// TIA Portal V20 program export: 7 tag tables, 10 data types, 12 data blocks, 14 code blocks (in call order from the OBs), 11 instance data blocks

VAR_GLOBAL   // PLC tag table "IO_PLC_Centralizer_PLC_Functinal_Test_1"
   In_Functional_Test_Odd AT %I100.0 : "IO_Device_Functinal_Test_Odd";
   Out_Test_Parameters_Odd AT %Q100.0 : "IO_Device_Test_Parameters_Odd";
   Voltage_Read_UInt AT %IW160 : UInt;
END_VAR

VAR_GLOBAL   // PLC tag table "IO_PLC_Centralizer_PLC_Functinal_Test_2"
   In_Functional_Test_Even AT %I300.0 : "IO_Device_Functinal_Test_Even";
   Out_Test_Parameters_Even AT %Q300.0 : "IO_Device_Test_Parameters_Even";
END_VAR

VAR_GLOBAL   // PLC tag table "IO_PLC_Centralizer_PLC_Functional_Test_Rework"
   In AT %I600.0 : "IO_Device_Functinal_Test_Rework";
   Out AT %Q600.0 : "IO_Device_Test_Parameters_Rework";
END_VAR

VAR_GLOBAL   // PLC tag table "PLC_Centralizer"
   Digital_Input_0 AT %I0.0 : Bool;
   Digital_Input_1 AT %I0.1 : Bool;
   Digital_Input_2 AT %I0.2 : Bool;
   Digital_Input_3 AT %I0.3 : Bool;
   Digital_Input_4 AT %I0.4 : Bool;
   Digital_Input_5 AT %I0.5 : Bool;
   Digital_Input_6 AT %I0.6 : Bool;
   Digital_Input_7 AT %I0.7 : Bool;
   Digital_Input_8 AT %I1.0 : Bool;
   Digital_Input_9 AT %I1.1 : Bool;
   Digital_Input_10 AT %I1.2 : Bool;
   Digital_Input_11 AT %I1.3 : Bool;
   Digital_Input_12 AT %I1.4 : Bool;
   Digital_Input_13 AT %I1.5 : Bool;
   Analogic_Input_0 AT %IW64 : Int;
   Analogic_Input_1 AT %IW66 : Int;
   Digital_Output_0 AT %Q0.0 : Bool;
   Digital_Output_1 AT %Q0.1 : Bool;
   Digital_Output_2 AT %Q0.2 : Bool;
   Digital_Output_3 AT %Q0.3 : Bool;
   Digital_Output_4 AT %Q0.4 : Bool;
   Digital_Output_5 AT %Q0.5 : Bool;
   Digital_Output_6 AT %Q0.6 : Bool;
   Digital_Output_7 AT %Q0.7 : Bool;
   Digital_Output_8 AT %Q1.0 : Bool;
   Digital_Output_9 AT %Q1.1 : Bool;
   Clock_Byte AT %MB0 : Byte;
   Clock_10Hz AT %M0.0 : Bool;
   Clock_5Hz AT %M0.1 : Bool;
   "Clock_2.5Hz" AT %M0.2 : Bool;
   Clock_2Hz AT %M0.3 : Bool;
   "Clock_1.25Hz" AT %M0.4 : Bool;
   Clock_1Hz AT %M0.5 : Bool;
   "Clock_0.625Hz" AT %M0.6 : Bool;
   "Clock_0.5Hz" AT %M0.7 : Bool;
   System_Byte AT %MB1 : Byte;
   FirstScan AT %M1.0 : Bool;
   DiagStatusUpdate AT %M1.1 : Bool;
   AlwaysTRUE AT %M1.2 : Bool;
   AlwaysFALSE AT %M1.3 : Bool;
END_VAR

VAR_GLOBAL   // PLC tag table "PLC_Centralizer_PLC_Production_And_Rework"
   In_PLC_Production_And_Rework AT %I500.0 : "IO_Device_Conveyor_Belt_Input";
   Out_PLC_Production_And_Rework AT %Q500.0 : "IO_Device_Conveyor_Belt_Ouput";
END_VAR

VAR_GLOBAL   // PLC tag table "SR-X100W_Entrace"
   Entrace_Read_Complete AT %I700.0 : Bool;
   Entrace_Read_Failure AT %I701.0 : Bool;
   Entrace_Read_Data AT %I702.0 : "SR-X100W_Read_Data";
   Entrace_Read_Request AT %Q700.0 : Bool;
   Entrace_Read_Complete_Clear AT %Q701.0 : Bool;
END_VAR

VAR_GLOBAL   // PLC tag table "SR-X100W_Exit"
   Exit_Read_Complete AT %I858.0 : Bool;
   Exit_Read_Failure AT %I859.0 : Bool;
   Exit_Read_Data AT %I860.0 : "SR-X100W_Read_Data";
   Exit_Read_Request AT %Q858.0 : Bool;
   Exit_Read_Complete_Clear AT %Q859.0 : Bool;
END_VAR

TYPE "Functional_Test"
   STRUCT
      Water_Fountain : String;
      Serial_Number : String[17];
      Panel_Number : SInt;
      Read_Electrical_Voltage : UInt;
      Read_Electrical_Current : UInt;
      Electrical_Current_Test : String[10];
      Visual_Test : String[10];
      Functional_Test : String[10];
   END_STRUCT;
END_TYPE

TYPE "IO_Device_Conveyor_Belt_Input"
   STRUCT
      Life_Trigger : Bool;
      Emergency_Stop_Release : Bool;
      Trigger_Read_Serial_Number_Entrace_Functional_Test : Bool;
      Trigger_Read_Serial_Number_Exit_Functional_Test : Bool;
      Selected_Voltage_220V : Bool;
      Selected_Voltage_127V : Bool;
      Carousel_Frequency_Inverter_Fail : Bool;
      Conveyor_Belt_Functional_Test_Inverter_Fail : Bool;
   END_STRUCT;
END_TYPE

TYPE "IO_Device_Conveyor_Belt_Ouput"
   STRUCT
      Start : Bool;
      Manual_Turn_On_Motor_Caroussel : Bool;
      Manual_Turn_On_Motor_Conveyor_Belt : Bool;
      Water_Foutain_Fail_Functional_Test : Bool;
      Select_Motor_Speed : SInt;
      Carousel_Voltage_Selection : SInt;
   END_STRUCT;
END_TYPE

TYPE "IO_Device_Functinal_Test_Even"
   STRUCT
      Life_Trigger_PLC_Functional_Test_2 : Bool;
      Star_Test_PLC_Functional_Test_2 : Bool;
      Button_PLC_Functional_Test_2 : Bool;
      Electrical_Current_Test_Approved_PLC_Functional_Test_2 : Bool;
      Visual_Test_Approved_PLC_Functional_Test_2 : Bool;
      Electrical_Current_Read_PLC_Functional_Test_2 : UInt;
      Life_Trigger_PLC_Functional_Test_4 : Bool;
      Star_Test_PLC_Functional_Test_4 : Bool;
      Button_PLC_Functional_Test_4 : Bool;
      Electrical_Current_Test_Approved_PLC_Functional_Test_4 : Bool;
      Visual_Test_Approved_PLC_Functional_Test_4 : Bool;
      Electrical_Current_Read_PLC_Functional_Test_4 : UInt;
      Life_Trigger_PLC_Functional_Test_6 : Bool;
      Star_Test_PLC_Functional_Test_6 : Bool;
      Button_PLC_Functional_Test_6 : Bool;
      Electrical_Current_Test_Approved_PLC_Functional_Test_6 : Bool;
      Visual_Test_Approved_PLC_Functional_Test_6 : Bool;
      Electrical_Current_Read_PLC_Functional_Test_6 : UInt;
      Life_Trigger_PLC_Functional_Test_8 : Bool;
      Star_Test_PLC_Functional_Test_8 : Bool;
      Button_PLC_Functional_Test_8 : Bool;
      Electrical_Current_Test_Approved_PLC_Functional_Test_8 : Bool;
      Visual_Test_Approved_PLC_Functional_Test_8 : Bool;
      Electrical_Current_Read_PLC_Functional_Test_8 : UInt;
      Life_Trigger_PLC_Functional_Test_10 : Bool;
      Star_Test_PLC_Functional_Test_10 : Bool;
      Button_PLC_Functional_Test_10 : Bool;
      Electrical_Current_Test_Approved_PLC_Functional_Test_10 : Bool;
      Visual_Test_Approved_PLC_Functional_Test_10 : Bool;
      Electrical_Current_Read_PLC_Functional_Test_10 : UInt;
      Life_Trigger_PLC_Functional_Test_12 : Bool;
      Star_Test_PLC_Functional_Test_12 : Bool;
      Button_PLC_Functional_Test_12 : Bool;
      Electrical_Current_Test_Approved_PLC_Functional_Test_12 : Bool;
      Visual_Test_Approved_PLC_Functional_Test_12 : Bool;
      Electrical_Current_Read_PLC_Functional_Test_12 : UInt;
      Life_Trigger_PLC_Functional_Test_14 : Bool;
      Star_Test_PLC_Functional_Test_14 : Bool;
      Button_PLC_Functional_Test_14 : Bool;
      Electrical_Current_Test_Approved_PLC_Functional_Test_14 : Bool;
      Visual_Test_Approved_PLC_Functional_Test_14 : Bool;
      Electrical_Current_Read_PLC_Functional_Test_14 : UInt;
      Life_Trigger_PLC_Functional_Test_16 : Bool;
      Star_Test_PLC_Functional_Test_16 : Bool;
      Button_PLC_Functional_Test_16 : Bool;
      Electrical_Current_Test_Approved_PLC_Functional_Test_16 : Bool;
      Visual_Test_Approved_PLC_Functional_Test_16 : Bool;
      Electrical_Current_Read_PLC_Functional_Test_16 : UInt;
      Life_Trigger_PLC_Functional_Test_18 : Bool;
      Star_Test_PLC_Functional_Test_18 : Bool;
      Button_PLC_Functional_Test_18 : Bool;
      Electrical_Current_Test_Approved_PLC_Functional_Test_18 : Bool;
      Visual_Test_Approved_PLC_Functional_Test_18 : Bool;
      Electrical_Current_Read_PLC_Functional_Test_18 : UInt;
      Life_Trigger_PLC_Functional_Test_20 : Bool;
      Star_Test_PLC_Functional_Test_20 : Bool;
      Button_PLC_Functional_Test_20 : Bool;
      Electrical_Current_Test_Approved_PLC_Functional_Test_20 : Bool;
      Visual_Test_Approved_PLC_Functional_Test_20 : Bool;
      Electrical_Current_Read_PLC_Functional_Test_20 : UInt;
      Life_Trigger_PLC_Functional_Test_22 : Bool;
      Star_Test_PLC_Functional_Test_22 : Bool;
      Button_PLC_Functional_Test_22 : Bool;
      Electrical_Current_Test_Approved_PLC_Functional_Test_22 : Bool;
      Visual_Test_Approved_PLC_Functional_Test_22 : Bool;
      Electrical_Current_Read_PLC_Functional_Test_22 : UInt;
      Life_Trigger_PLC_Functional_Test_24 : Bool;
      Star_Test_PLC_Functional_Test_24 : Bool;
      Button_PLC_Functional_Test_24 : Bool;
      Electrical_Current_Test_Approved_PLC_Functional_Test_24 : Bool;
      Visual_Test_Approved_PLC_Functional_Test_24 : Bool;
      Electrical_Current_Read_PLC_Functional_Test_24 : UInt;
      Life_Trigger_PLC_Functional_Test_26 : Bool;
      Star_Test_PLC_Functional_Test_26 : Bool;
      Button_PLC_Functional_Test_26 : Bool;
      Electrical_Current_Test_Approved_PLC_Functional_Test_26 : Bool;
      Visual_Test_Approved_PLC_Functional_Test_26 : Bool;
      Electrical_Current_Read_PLC_Functional_Test_26 : UInt;
      Life_Trigger_PLC_Functional_Test_28 : Bool;
      Star_Test_PLC_Functional_Test_28 : Bool;
      Button_PLC_Functional_Test_28 : Bool;
      Electrical_Current_Test_Approved_PLC_Functional_Test_28 : Bool;
      Visual_Test_Approved_PLC_Functional_Test_28 : Bool;
      Electrical_Current_Read_PLC_Functional_Test_28 : UInt;
      Life_Trigger_PLC_Functional_Test_30 : Bool;
      Star_Test_PLC_Functional_Test_30 : Bool;
      Button_PLC_Functional_Test_30 : Bool;
      Electrical_Current_Test_Approved_PLC_Functional_Test_30 : Bool;
      Visual_Test_Approved_PLC_Functional_Test_30 : Bool;
      Electrical_Current_Read_PLC_Functional_Test_30 : UInt;
   END_STRUCT;
END_TYPE

TYPE "IO_Device_Functinal_Test_Odd"
   STRUCT
      Life_Trigger_PLC_Functional_Test_1 : Bool;
      Star_Test_PLC_Functional_Test_1 : Bool;
      Button_PLC_Functional_Test_1 : Bool;
      Electrical_Current_Test_Approved_PLC_Functional_Test_1 : Bool;
      Visual_Test_Approved_PLC_Functional_Test_1 : Bool;
      Electrical_Current_Read_PLC_Functional_Test_1 : UInt;
      Life_Trigger_PLC_Functional_Test_3 : Bool;
      Star_Test_PLC_Functional_Test_3 : Bool;
      Button_PLC_Functional_Test_3 : Bool;
      Electrical_Current_Test_Approved_PLC_Functional_Test_3 : Bool;
      Visual_Test_Approved_PLC_Functional_Test_3 : Bool;
      Electrical_Current_Read_PLC_Functional_Test_3 : UInt;
      Life_Trigger_PLC_Functional_Test_5 : Bool;
      Star_Test_PLC_Functional_Test_5 : Bool;
      Button_PLC_Functional_Test_5 : Bool;
      Electrical_Current_Test_Approved_PLC_Functional_Test_5 : Bool;
      Visual_Test_Approved_PLC_Functional_Test_5 : Bool;
      Electrical_Current_Read_PLC_Functional_Test_5 : UInt;
      Life_Trigger_PLC_Functional_Test_7 : Bool;
      Star_Test_PLC_Functional_Test_7 : Bool;
      Button_PLC_Functional_Test_7 : Bool;
      Electrical_Current_Test_Approved_PLC_Functional_Test_7 : Bool;
      Visual_Test_Approved_PLC_Functional_Test_7 : Bool;
      Electrical_Current_Read_PLC_Functional_Test_7 : UInt;
      Life_Trigger_PLC_Functional_Test_9 : Bool;
      Star_Test_PLC_Functional_Test_9 : Bool;
      Button_PLC_Functional_Test_9 : Bool;
      Electrical_Current_Test_Approved_PLC_Functional_Test_9 : Bool;
      Visual_Test_Approved_PLC_Functional_Test_9 : Bool;
      Electrical_Current_Read_PLC_Functional_Test_9 : UInt;
      Life_Trigger_PLC_Functional_Test_11 : Bool;
      Star_Test_PLC_Functional_Test_11 : Bool;
      Button_PLC_Functional_Test_11 : Bool;
      Electrical_Current_Test_Approved_PLC_Functional_Test_11 : Bool;
      Visual_Test_Approved_PLC_Functional_Test_11 : Bool;
      Electrical_Current_Read_PLC_Functional_Test_11 : UInt;
      Life_Trigger_PLC_Functional_Test_13 : Bool;
      Star_Test_PLC_Functional_Test_13 : Bool;
      Button_PLC_Functional_Test_13 : Bool;
      Electrical_Current_Test_Approved_PLC_Functional_Test_13 : Bool;
      Visual_Test_Approved_PLC_Functional_Test_13 : Bool;
      Electrical_Current_Read_PLC_Functional_Test_13 : UInt;
      Life_Trigger_PLC_Functional_Test_15 : Bool;
      Star_Test_PLC_Functional_Test_15 : Bool;
      Button_PLC_Functional_Test_15 : Bool;
      Electrical_Current_Test_Approved_PLC_Functional_Test_15 : Bool;
      Visual_Test_Approved_PLC_Functional_Test_15 : Bool;
      Electrical_Current_Read_PLC_Functional_Test_15 : UInt;
      Life_Trigger_PLC_Functional_Test_17 : Bool;
      Star_Test_PLC_Functional_Test_17 : Bool;
      Button_PLC_Functional_Test_17 : Bool;
      Electrical_Current_Test_Approved_PLC_Functional_Test_17 : Bool;
      Visual_Test_Approved_PLC_Functional_Test_17 : Bool;
      Electrical_Current_Read_PLC_Functional_Test_17 : UInt;
      Life_Trigger_PLC_Functional_Test_19 : Bool;
      Star_Test_PLC_Functional_Test_19 : Bool;
      Button_PLC_Functional_Test_19 : Bool;
      Electrical_Current_Test_Approved_PLC_Functional_Test_19 : Bool;
      Visual_Test_Approved_PLC_Functional_Test_19 : Bool;
      Electrical_Current_Read_PLC_Functional_Test_19 : UInt;
      Life_Trigger_PLC_Functional_Test_21 : Bool;
      Star_Test_PLC_Functional_Test_21 : Bool;
      Button_PLC_Functional_Test_21 : Bool;
      Electrical_Current_Test_Approved_PLC_Functional_Test_21 : Bool;
      Visual_Test_Approved_PLC_Functional_Test_21 : Bool;
      Electrical_Current_Read_PLC_Functional_Test_21 : UInt;
      Life_Trigger_PLC_Functional_Test_23 : Bool;
      Star_Test_PLC_Functional_Test_23 : Bool;
      Button_PLC_Functional_Test_23 : Bool;
      Electrical_Current_Test_Approved_PLC_Functional_Test_23 : Bool;
      Visual_Test_Approved_PLC_Functional_Test_23 : Bool;
      Electrical_Current_Read_PLC_Functional_Test_23 : UInt;
      Life_Trigger_PLC_Functional_Test_25 : Bool;
      Star_Test_PLC_Functional_Test_25 : Bool;
      Button_PLC_Functional_Test_25 : Bool;
      Electrical_Current_Test_Approved_PLC_Functional_Test_25 : Bool;
      Visual_Test_Approved_PLC_Functional_Test_25 : Bool;
      Electrical_Current_Read_PLC_Functional_Test_25 : UInt;
      Life_Trigger_PLC_Functional_Test_27 : Bool;
      Star_Test_PLC_Functional_Test_27 : Bool;
      Button_PLC_Functional_Test_27 : Bool;
      Electrical_Current_Test_Approved_PLC_Functional_Test_27 : Bool;
      Visual_Test_Approved_PLC_Functional_Test_27 : Bool;
      Electrical_Current_Read_PLC_Functional_Test_27 : UInt;
      Life_Trigger_PLC_Functional_Test_29 : Bool;
      Star_Test_PLC_Functional_Test_29 : Bool;
      Button_PLC_Functional_Test_29 : Bool;
      Electrical_Current_Test_Approved_PLC_Functional_Test_29 : Bool;
      Visual_Test_Approved_PLC_Functional_Test_29 : Bool;
      Electrical_Current_Read_PLC_Functional_Test_29 : UInt;
   END_STRUCT;
END_TYPE

TYPE "IO_Device_Functinal_Test_Rework"
   STRUCT
      Life_Trigger_PLC_Functional_Test_Rework : Bool;
      Star_Test_PLC_Functional_Test_Rework : Bool;
      Button_PLC_Functional_Test_Rework : Bool;
      Electrical_Current_Test_Approved_PLC_Functional_Test_Rework : Bool;
      Visual_Test_Approved_PLC_Functional_Test_Rework : Bool;
      Electrical_Current_Read_PLC_Functional_Test_Rework : UInt;
   END_STRUCT;
END_TYPE

TYPE "IO_Device_Test_Parameters_Even"
   STRUCT
      Reset_PLC_Functional_Test_2 : Bool;
      Reset_PLC_Functional_Test_4 : Bool;
      Reset_PLC_Functional_Test_6 : Bool;
      Reset_PLC_Functional_Test_8 : Bool;
      Reset_PLC_Functional_Test_10 : Bool;
      Reset_PLC_Functional_Test_12 : Bool;
      Reset_PLC_Functional_Test_14 : Bool;
      Reset_PLC_Functional_Test_16 : Bool;
      Reset_PLC_Functional_Test_18 : Bool;
      Reset_PLC_Functional_Test_20 : Bool;
      Reset_PLC_Functional_Test_22 : Bool;
      Reset_PLC_Functional_Test_24 : Bool;
      Reset_PLC_Functional_Test_26 : Bool;
      Reset_PLC_Functional_Test_28 : Bool;
      Reset_PLC_Functional_Test_30 : Bool;
      Status : Bool;
      Voltage_Read : UInt;
      Min_Electrical_Current : UInt;
      Max_Electrical_Current : UInt;
      Time_End_Electrical_Current_Test : Time;
      Time_Start_Visual_Test : Time;
   END_STRUCT;
END_TYPE

TYPE "IO_Device_Test_Parameters_Odd"
   STRUCT
      Reset_PLC_Functional_Test_1 : Bool;
      Reset_PLC_Functional_Test_3 : Bool;
      Reset_PLC_Functional_Test_5 : Bool;
      Reset_PLC_Functional_Test_7 : Bool;
      Reset_PLC_Functional_Test_9 : Bool;
      Reset_PLC_Functional_Test_11 : Bool;
      Reset_PLC_Functional_Test_13 : Bool;
      Reset_PLC_Functional_Test_15 : Bool;
      Reset_PLC_Functional_Test_17 : Bool;
      Reset_PLC_Functional_Test_19 : Bool;
      Reset_PLC_Functional_Test_21 : Bool;
      Reset_PLC_Functional_Test_23 : Bool;
      Reset_PLC_Functional_Test_25 : Bool;
      Reset_PLC_Functional_Test_27 : Bool;
      Reset_PLC_Functional_Test_29 : Bool;
      Status : Bool;
      Voltage_Read : UInt;
      Min_Electrical_Current : UInt;
      Max_Electrical_Current : UInt;
      Time_End_Electrical_Current_Test : Time;
      Time_Start_Visual_Test : Time;
   END_STRUCT;
END_TYPE

TYPE "IO_Device_Test_Parameters_Rework"
   STRUCT
      Reset_PLC_Functional_Test_Rework : Bool;
      Status : Bool;
      Voltage_Read : UInt;
      Min_Electrical_Current : UInt;
      Max_Electrical_Current : UInt;
      Time_End_Electrical_Current_Test : Time;
      Time_Start_Visual_Test : Time;
   END_STRUCT;
END_TYPE

TYPE "SR-X100W_Read_Data"
   STRUCT
      "sr-x_100_Read_Data_1" : Char;
      "sr-x_100_Read_Data_2" : Char;
      "sr-x_100_Read_Data_3" : Char;
      "sr-x_100_Read_Data_4" : Char;
      "sr-x_100_Read_Data_5" : Char;
      "sr-x_100_Read_Data_6" : Char;
      "sr-x_100_Read_Data_7" : Char;
      "sr-x_100_Read_Data_8" : Char;
      "sr-x_100_Read_Data_9" : Char;
      "sr-x_100_Read_Data_10" : Char;
      "sr-x_100_Read_Data_11" : Char;
      "sr-x_100_Read_Data_12" : Char;
      "sr-x_100_Read_Data_13" : Char;
      "sr-x_100_Read_Data_14" : Char;
      "sr-x_100_Read_Data_15" : Char;
      "sr-x_100_Read_Data_16" : Char;
      "sr-x_100_Read_Data_17" : Char;
      "sr-x_100_Read_Data_18" : Char;
      "sr-x_100_Read_Data_19" : Char;
      "sr-x_100_Read_Data_20" : Char;
      "sr-x_100_Read_Data_21" : Char;
      "sr-x_100_Read_Data_22" : Char;
      "sr-x_100_Read_Data_23" : Char;
      "sr-x_100_Read_Data_24" : Char;
      "sr-x_100_Read_Data_25" : Char;
      "sr-x_100_Read_Data_26" : Char;
      "sr-x_100_Read_Data_27" : Char;
      "sr-x_100_Read_Data_28" : Char;
      "sr-x_100_Read_Data_29" : Char;
      "sr-x_100_Read_Data_30" : Char;
      "sr-x_100_Read_Data_31" : Char;
      "sr-x_100_Read_Data_32" : Char;
      "sr-x_100_Read_Data_33" : Char;
      "sr-x_100_Read_Data_34" : Char;
      "sr-x_100_Read_Data_35" : Char;
      "sr-x_100_Read_Data_36" : Char;
      "sr-x_100_Read_Data_37" : Char;
      "sr-x_100_Read_Data_38" : Char;
      "sr-x_100_Read_Data_39" : Char;
      "sr-x_100_Read_Data_40" : Char;
      "sr-x_100_Read_Data_41" : Char;
      "sr-x_100_Read_Data_42" : Char;
      "sr-x_100_Read_Data_43" : Char;
      "sr-x_100_Read_Data_44" : Char;
      "sr-x_100_Read_Data_45" : Char;
      "sr-x_100_Read_Data_46" : Char;
      "sr-x_100_Read_Data_47" : Char;
      "sr-x_100_Read_Data_48" : Char;
      "sr-x_100_Read_Data_49" : Char;
      "sr-x_100_Read_Data_50" : Char;
      "sr-x_100_Read_Data_51" : Char;
      "sr-x_100_Read_Data_52" : Char;
      "sr-x_100_Read_Data_53" : Char;
      "sr-x_100_Read_Data_54" : Char;
      "sr-x_100_Read_Data_55" : Char;
      "sr-x_100_Read_Data_56" : Char;
      "sr-x_100_Read_Data_57" : Char;
      "sr-x_100_Read_Data_58" : Char;
      "sr-x_100_Read_Data_59" : Char;
      "sr-x_100_Read_Data_60" : Char;
      "sr-x_100_Read_Data_61" : Char;
      "sr-x_100_Read_Data_62" : Char;
      "sr-x_100_Read_Data_63" : Char;
      "sr-x_100_Read_Data_64" : Char;
      "sr-x_100_Read_Data_65" : Char;
      "sr-x_100_Read_Data_66" : Char;
      "sr-x_100_Read_Data_67" : Char;
      "sr-x_100_Read_Data_68" : Char;
      "sr-x_100_Read_Data_69" : Char;
      "sr-x_100_Read_Data_70" : Char;
      "sr-x_100_Read_Data_71" : Char;
      "sr-x_100_Read_Data_72" : Char;
      "sr-x_100_Read_Data_73" : Char;
      "sr-x_100_Read_Data_74" : Char;
      "sr-x_100_Read_Data_75" : Char;
      "sr-x_100_Read_Data_76" : Char;
      "sr-x_100_Read_Data_77" : Char;
      "sr-x_100_Read_Data_78" : Char;
      "sr-x_100_Read_Data_79" : Char;
      "sr-x_100_Read_Data_80" : Char;
      "sr-x_100_Read_Data_81" : Char;
      "sr-x_100_Read_Data_82" : Char;
      "sr-x_100_Read_Data_83" : Char;
      "sr-x_100_Read_Data_84" : Char;
      "sr-x_100_Read_Data_85" : Char;
      "sr-x_100_Read_Data_86" : Char;
      "sr-x_100_Read_Data_87" : Char;
      "sr-x_100_Read_Data_88" : Char;
      "sr-x_100_Read_Data_89" : Char;
      "sr-x_100_Read_Data_90" : Char;
      "sr-x_100_Read_Data_91" : Char;
      "sr-x_100_Read_Data_92" : Char;
      "sr-x_100_Read_Data_93" : Char;
      "sr-x_100_Read_Data_94" : Char;
      "sr-x_100_Read_Data_95" : Char;
      "sr-x_100_Read_Data_96" : Char;
      "sr-x_100_Read_Data_97" : Char;
      "sr-x_100_Read_Data_98" : Char;
      "sr-x_100_Read_Data_99" : Char;
      "sr-x_100_Read_Data_100" : Char;
      "sr-x_100_Read_Data_101" : Char;
      "sr-x_100_Read_Data_102" : Char;
      "sr-x_100_Read_Data_103" : Char;
      "sr-x_100_Read_Data_104" : Char;
      "sr-x_100_Read_Data_105" : Char;
      "sr-x_100_Read_Data_106" : Char;
      "sr-x_100_Read_Data_107" : Char;
      "sr-x_100_Read_Data_108" : Char;
      "sr-x_100_Read_Data_109" : Char;
      "sr-x_100_Read_Data_110" : Char;
      "sr-x_100_Read_Data_111" : Char;
      "sr-x_100_Read_Data_112" : Char;
      "sr-x_100_Read_Data_113" : Char;
      "sr-x_100_Read_Data_114" : Char;
      "sr-x_100_Read_Data_115" : Char;
      "sr-x_100_Read_Data_116" : Char;
      "sr-x_100_Read_Data_117" : Char;
      "sr-x_100_Read_Data_118" : Char;
      "sr-x_100_Read_Data_119" : Char;
      "sr-x_100_Read_Data_120" : Char;
      "sr-x_100_Read_Data_121" : Char;
      "sr-x_100_Read_Data_122" : Char;
      "sr-x_100_Read_Data_123" : Char;
      "sr-x_100_Read_Data_124" : Char;
      "sr-x_100_Read_Data_125" : Char;
      "sr-x_100_Read_Data_126" : Char;
      "sr-x_100_Read_Data_127" : Char;
      "sr-x_100_Read_Data_128" : Char;
      "sr-x_100_Read_Data_129" : Char;
      "sr-x_100_Read_Data_130" : Char;
      "sr-x_100_Read_Data_131" : Char;
      "sr-x_100_Read_Data_132" : Char;
      "sr-x_100_Read_Data_133" : Char;
      "sr-x_100_Read_Data_134" : Char;
      "sr-x_100_Read_Data_135" : Char;
      "sr-x_100_Read_Data_136" : Char;
   END_STRUCT;
END_TYPE

DATA_BLOCK "DB_Analogic_Inputs"   // DB2
{ S7_Optimized_Access := 'TRUE' }
// stored: MemoryReserve 100
   VAR
      Real_Analogic_Input_0 : Real;
      Real_Analogic_Input_1 : Real;
      Uint_Analogic_Input_0 : UInt;
      Uint_Analogic_Input_1 : UInt;
   END_VAR
BEGIN
END_DATA_BLOCK

DATA_BLOCK "DB_DataLog"   // DB12
{ S7_Optimized_Access := 'TRUE' }
// stored: MemoryReserve 100
   VAR
      Create_DataLog : Bool;
      Open_DataLog : Bool;
      Write_DataLog : Bool;
      Close_DataLog : Bool;
      Clean_DataLog : Bool;
      Delete_DataLog : Bool;
      ID_DataLog : DWord;
      Name_DataLog : String := 'Teste Funcional';
      Header_DataLog : String := 'Bebedoro,Numero de Serie,Painel,Tensao Eletrica [V],Corrente Eletrica [mA],Resultado Teste Corrente,Resultado Teste Visual,Resultado Teste Funcional';
   END_VAR
BEGIN
END_DATA_BLOCK

DATA_BLOCK "DB_Digital_Inputs"   // DB1
{ S7_Optimized_Access := 'TRUE' }
// stored: MemoryReserve 100
   VAR
      Digital_Input_0 : Bool;
      Digital_Input_1 : Bool;
      Digital_Input_2 : Bool;
      Digital_Input_3 : Bool;
      Digital_Input_4 : Bool;
      Digital_Input_5 : Bool;
      Digital_Input_6 : Bool;
      Digital_Input_7 : Bool;
      Digital_Input_8 : Bool;
      Digital_Input_9 : Bool;
      Digital_Input_10 : Bool;
      Digital_Input_11 : Bool;
      Digital_Input_12 : Bool;
      Digital_Input_13 : Bool;
   END_VAR
BEGIN
END_DATA_BLOCK

DATA_BLOCK "DB_Digital_Outputs"   // DB3
{ S7_Optimized_Access := 'TRUE' }
// stored: MemoryReserve 100
   VAR
      Digital_Output_0 : Bool;
      Digital_Output_1 : Bool;
      Digital_Output_2 : Bool;
      Digital_Output_3 : Bool;
      Digital_Output_4 : Bool;
      Digital_Output_5 : Bool;
      Digital_Output_6 : Bool;
      Digital_Output_7 : Bool;
      Digital_Output_8 : Bool;
      Digital_Output_9 : Bool;
   END_VAR
BEGIN
END_DATA_BLOCK

DATA_BLOCK "DB_Found_Water_Fountain_Functional_Test"   // DB11
{ S7_Optimized_Access := 'TRUE' }
// stored: MemoryReserve 100
   VAR
      Found_Functional_Test : Bool;
      Water_Foutain_Fail_Functional_Test : Bool;
      i : SInt;
      Water_Foutain_Functional_Test : "Functional_Test";
   END_VAR
BEGIN
END_DATA_BLOCK

DATA_BLOCK "DB_HMI"   // DB4
{ S7_Optimized_Access := 'TRUE' }
// stored: MemoryReserve 100
   VAR
      Job_Mailbox : Array[0..3] of Word;
      Control_Screen : Word := 1;
      Alarm : Bool;
      Start : Bool;
      Change_Employee : Bool;
      Send_Recipe : Bool;
      Manual_Turn_On_Motor_Caroussel : Bool;
      Manual_Turn_On_Motor_Conveyor_Belt : Bool;
      Select_Test_Panel : SInt;
      Select_Motor_Speed : SInt := 1;
      Employee_Rework : String[6];
      Employee_Station_1 : String[6];
      Employee_Station_2 : String[6];
   END_VAR
   VAR RETAIN
      Admin_1 : String[6];
      Admin_2 : String[6];
      Admin_3 : String[6];
      Admin_4 : String[6];
      Admin_5 : String[6];
   END_VAR
   VAR
      Serial_Number : String[17];
      Electrical_Current : UInt;
      Electrical_Voltage : UInt;
      Electrical_Current_Result : String[10];
      Visual_Test_Result : String[10];
      Functional_Test_Result : String[10];
      Rework_Serial_Number : String[17];
      Rework_Electrical_Current : UInt;
      Rework_Electrical_Voltage : UInt;
      Rework_Electrical_Current_Result : String[10];
      Rework_Visual_Test_Result : String[10];
      Rework_Functional_Test_Result : String[10];
      Alarm_0 : Word;
      Alarm_1 : Word;
      Alarm_2 : Word;
   END_VAR
BEGIN
END_DATA_BLOCK

DATA_BLOCK "DB_IO_Device_In_Functional_Test"   // DB6
{ S7_Optimized_Access := 'TRUE' }
// stored: MemoryReserve 100
   VAR
      Reset_PLC_Functional_Test : Array[0..31] of Bool;
      Status : Bool;
      Voltage_Read : UInt;
   END_VAR
BEGIN
END_DATA_BLOCK

DATA_BLOCK "DB_IO_Device_In_Production and Rework"   // DB7
{ S7_Optimized_Access := 'TRUE' }
// stored: AutoNumber false, MemoryReserve 100
   VAR
      Emergency_Stop_Release : Bool;
      Trigger_Read_Serial_Number_Entrace_Functional_Test : Bool;
      Trigger_Read_Serial_Number_Exit_Functional_Test : Bool;
      Selected_Voltage_220V : Bool;
      Selected_Voltage_127V : Bool;
      Carousel_Frequency_Inverter_Fail : Bool;
      Conveyor_Belt_Functional_Test_Inverter_Fail : Bool;
   END_VAR
BEGIN
END_DATA_BLOCK

DATA_BLOCK "DB_Marrige"   // DB10
{ S7_Optimized_Access := 'TRUE' }
// stored: AutoNumber false, MemoryReserve 100
   VAR
      Functional_Tests_Panels : Array[0..31] of "Functional_Test";
      Got_Married { S7_SetPoint := 'True'} : Bool;
      Serial_Number : String[17];
   END_VAR
BEGIN
   Functional_Tests_Panels[0].Panel_Number := 0;
   Functional_Tests_Panels[1].Panel_Number := 1;
   Functional_Tests_Panels[2].Panel_Number := 2;
   Functional_Tests_Panels[3].Panel_Number := 3;
   Functional_Tests_Panels[4].Panel_Number := 4;
   Functional_Tests_Panels[5].Panel_Number := 5;
   Functional_Tests_Panels[6].Panel_Number := 6;
   Functional_Tests_Panels[7].Panel_Number := 7;
   Functional_Tests_Panels[8].Panel_Number := 8;
   Functional_Tests_Panels[9].Panel_Number := 9;
   Functional_Tests_Panels[10].Panel_Number := 10;
   Functional_Tests_Panels[11].Panel_Number := 11;
   Functional_Tests_Panels[12].Panel_Number := 12;
   Functional_Tests_Panels[13].Panel_Number := 13;
   Functional_Tests_Panels[14].Panel_Number := 14;
   Functional_Tests_Panels[15].Panel_Number := 15;
   Functional_Tests_Panels[16].Panel_Number := 16;
   Functional_Tests_Panels[17].Panel_Number := 17;
   Functional_Tests_Panels[18].Panel_Number := 18;
   Functional_Tests_Panels[19].Panel_Number := 19;
   Functional_Tests_Panels[20].Panel_Number := 20;
   Functional_Tests_Panels[21].Panel_Number := 21;
   Functional_Tests_Panels[22].Panel_Number := 22;
   Functional_Tests_Panels[23].Panel_Number := 23;
   Functional_Tests_Panels[24].Panel_Number := 24;
   Functional_Tests_Panels[25].Panel_Number := 25;
   Functional_Tests_Panels[26].Panel_Number := 26;
   Functional_Tests_Panels[27].Panel_Number := 27;
   Functional_Tests_Panels[28].Panel_Number := 28;
   Functional_Tests_Panels[29].Panel_Number := 29;
   Functional_Tests_Panels[30].Panel_Number := 30;
   Functional_Tests_Panels[31].Panel_Number := 31;
END_DATA_BLOCK

DATA_BLOCK "DB_Recipe"   // DB5
{ S7_Optimized_Access := 'TRUE' }
// stored: MemoryReserve 100
   VAR
      Water_Fountain : String;
      Voltage : SInt;
      Min_Electrical_Current : UInt;
      Max_Electrical_Current : UInt;
      Time_End_Electrical_Current_Test : Time;
      Time_Start_Visual_Test : Time;
   END_VAR
BEGIN
END_DATA_BLOCK

DATA_BLOCK "DB_SR-X100W_Entrace"   // DB8
{ S7_Optimized_Access := 'TRUE' }
// stored: MemoryReserve 100
   VAR
      Read_Complete_OUT : Bool;
      Read_Failure_OUT : Bool;
      Read_Data_Out : String[136];
      Serial_Number : String[17];
   END_VAR
BEGIN
END_DATA_BLOCK

DATA_BLOCK "DB_SR-X100W_Exit"   // DB9
{ S7_Optimized_Access := 'TRUE' }
// stored: AutoNumber false, MemoryReserve 100
   VAR
      Read_Complete_OUT : Bool;
      Read_Failure_OUT : Bool;
      Read_Data_Out : String[136];
      Serial_Number : String[17];
   END_VAR
BEGIN
END_DATA_BLOCK

ORGANIZATION_BLOCK "Main"   // OB1, LAD, ProgramCycle
TITLE = "Main Program Sweep (Cycle)"
{ S7_Optimized_Access := 'TRUE' }
// stored: SetENOAutomatically false
   VAR_INPUT
      Initial_Call : Bool;   // Initial call of this OB
      Remanence : Bool;   // =True, if remanent data are available
   END_VAR
BEGIN

REGION Network 1
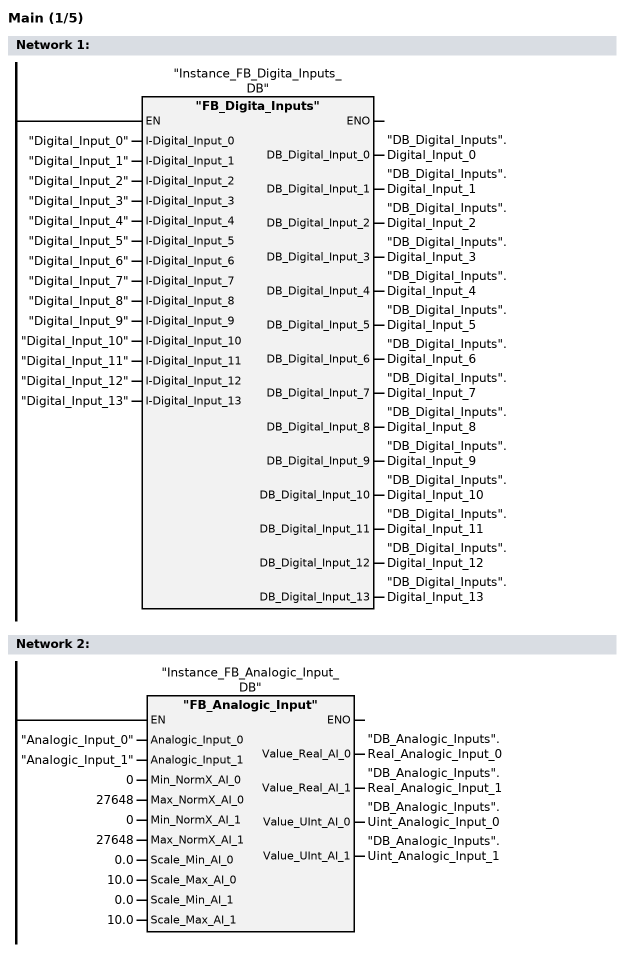
   RUNG wire#powerrail
      "Instance_FB_Digita_Inputs_DB"("I-Digital_Input_0" := "Digital_Input_0", "I-Digital_Input_1" := "Digital_Input_1", "I-Digital_Input_2" := "Digital_Input_2", "I-Digital_Input_3" := "Digital_Input_3", "I-Digital_Input_4" := "Digital_Input_4", "I-Digital_Input_5" := "Digital_Input_5", "I-Digital_Input_6" := "Digital_Input_6", "I-Digital_Input_7" := "Digital_Input_7", "I-Digital_Input_8" := "Digital_Input_8", "I-Digital_Input_9" := "Digital_Input_9", "I-Digital_Input_10" := "Digital_Input_10", "I-Digital_Input_11" := "Digital_Input_11", "I-Digital_Input_12" := "Digital_Input_12", "I-Digital_Input_13" := "Digital_Input_13", DB_Digital_Input_0 => "DB_Digital_Inputs".Digital_Input_0, DB_Digital_Input_1 => "DB_Digital_Inputs".Digital_Input_1, DB_Digital_Input_2 => "DB_Digital_Inputs".Digital_Input_2, DB_Digital_Input_3 => "DB_Digital_Inputs".Digital_Input_3, DB_Digital_Input_4 => "DB_Digital_Inputs".Digital_Input_4, DB_Digital_Input_5 => "DB_Digital_Inputs".Digital_Input_5, DB_Digital_Input_6 => "DB_Digital_Inputs".Digital_Input_6, DB_Digital_Input_7 => "DB_Digital_Inputs".Digital_Input_7, DB_Digital_Input_8 => "DB_Digital_Inputs".Digital_Input_8, DB_Digital_Input_9 => "DB_Digital_Inputs".Digital_Input_9, DB_Digital_Input_10 => "DB_Digital_Inputs".Digital_Input_10, DB_Digital_Input_11 => "DB_Digital_Inputs".Digital_Input_11, DB_Digital_Input_12 => "DB_Digital_Inputs".Digital_Input_12, DB_Digital_Input_13 => "DB_Digital_Inputs".Digital_Input_13)
   END_RUNG
   // the same network as SCL:
   "Instance_FB_Digita_Inputs_DB"("I-Digital_Input_0" := "Digital_Input_0",   // "FB_Digita_Inputs"
                           "I-Digital_Input_1" := "Digital_Input_1",
                           "I-Digital_Input_2" := "Digital_Input_2",
                           "I-Digital_Input_3" := "Digital_Input_3",
                           "I-Digital_Input_4" := "Digital_Input_4",
                           "I-Digital_Input_5" := "Digital_Input_5",
                           "I-Digital_Input_6" := "Digital_Input_6",
                           "I-Digital_Input_7" := "Digital_Input_7",
                           "I-Digital_Input_8" := "Digital_Input_8",
                           "I-Digital_Input_9" := "Digital_Input_9",
                           "I-Digital_Input_10" := "Digital_Input_10",
                           "I-Digital_Input_11" := "Digital_Input_11",
                           "I-Digital_Input_12" := "Digital_Input_12",
                           "I-Digital_Input_13" := "Digital_Input_13",
                           DB_Digital_Input_0 => "DB_Digital_Inputs".Digital_Input_0,
                           DB_Digital_Input_1 => "DB_Digital_Inputs".Digital_Input_1,
                           DB_Digital_Input_2 => "DB_Digital_Inputs".Digital_Input_2,
                           DB_Digital_Input_3 => "DB_Digital_Inputs".Digital_Input_3,
                           DB_Digital_Input_4 => "DB_Digital_Inputs".Digital_Input_4,
                           DB_Digital_Input_5 => "DB_Digital_Inputs".Digital_Input_5,
                           DB_Digital_Input_6 => "DB_Digital_Inputs".Digital_Input_6,
                           DB_Digital_Input_7 => "DB_Digital_Inputs".Digital_Input_7,
                           DB_Digital_Input_8 => "DB_Digital_Inputs".Digital_Input_8,
                           DB_Digital_Input_9 => "DB_Digital_Inputs".Digital_Input_9,
                           DB_Digital_Input_10 => "DB_Digital_Inputs".Digital_Input_10,
                           DB_Digital_Input_11 => "DB_Digital_Inputs".Digital_Input_11,
                           DB_Digital_Input_12 => "DB_Digital_Inputs".Digital_Input_12,
                           DB_Digital_Input_13 => "DB_Digital_Inputs".Digital_Input_13);
END_REGION

REGION Network 2
   RUNG wire#powerrail
      "Instance_FB_Analogic_Input_DB"(Analogic_Input_0 := "Analogic_Input_0", Analogic_Input_1 := "Analogic_Input_1", Min_NormX_AI_0 := 0, Max_NormX_AI_0 := 27648, Min_NormX_AI_1 := 0, Max_NormX_AI_1 := 27648, Scale_Min_AI_0 := 0.0, Scale_Max_AI_0 := 10.0, Scale_Min_AI_1 := 0.0, Scale_Max_AI_1 := 10.0, Value_Real_AI_0 => "DB_Analogic_Inputs".Real_Analogic_Input_0, Value_Real_AI_1 => "DB_Analogic_Inputs".Real_Analogic_Input_1, Value_UInt_AI_0 => "DB_Analogic_Inputs".Uint_Analogic_Input_0, Value_UInt_AI_1 => "DB_Analogic_Inputs".Uint_Analogic_Input_1)
   END_RUNG
   // the same network as SCL:
   "Instance_FB_Analogic_Input_DB"(Analogic_Input_0 := "Analogic_Input_0",   // "FB_Analogic_Input"
                           Analogic_Input_1 := "Analogic_Input_1",
                           Min_NormX_AI_0 := 0,
                           Max_NormX_AI_0 := 27648,
                           Min_NormX_AI_1 := 0,
                           Max_NormX_AI_1 := 27648,
                           Scale_Min_AI_0 := 0.0,
                           Scale_Max_AI_0 := 10.0,
                           Scale_Min_AI_1 := 0.0,
                           Scale_Max_AI_1 := 10.0,
                           Value_Real_AI_0 => "DB_Analogic_Inputs".Real_Analogic_Input_0,
                           Value_Real_AI_1 => "DB_Analogic_Inputs".Real_Analogic_Input_1,
                           Value_UInt_AI_0 => "DB_Analogic_Inputs".Uint_Analogic_Input_0,
                           Value_UInt_AI_1 => "DB_Analogic_Inputs".Uint_Analogic_Input_1);
END_REGION

REGION Network 3
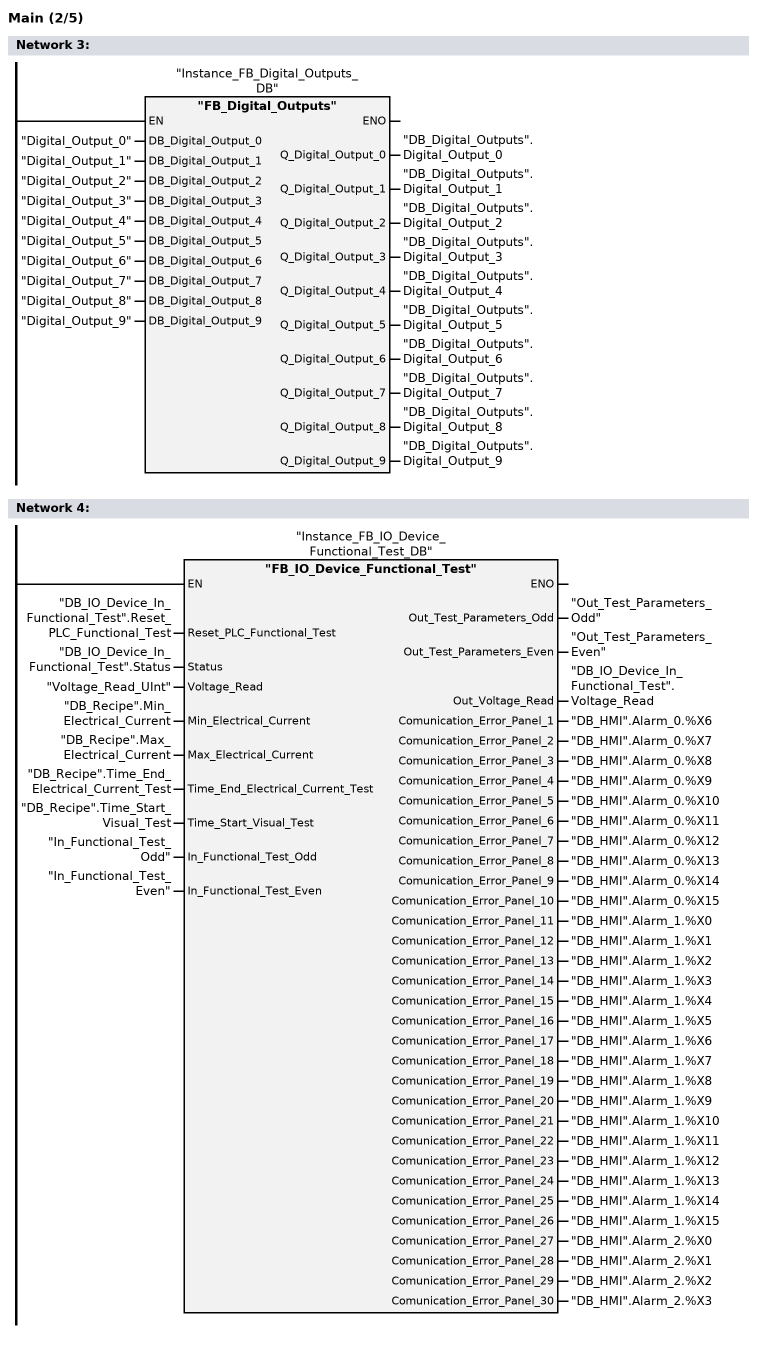
   RUNG wire#powerrail
      "Instance_FB_Digital_Outputs_DB"(DB_Digital_Output_0 := "Digital_Output_0", DB_Digital_Output_1 := "Digital_Output_1", DB_Digital_Output_2 := "Digital_Output_2", DB_Digital_Output_3 := "Digital_Output_3", DB_Digital_Output_4 := "Digital_Output_4", DB_Digital_Output_5 := "Digital_Output_5", DB_Digital_Output_6 := "Digital_Output_6", DB_Digital_Output_7 := "Digital_Output_7", DB_Digital_Output_8 := "Digital_Output_8", DB_Digital_Output_9 := "Digital_Output_9", Q_Digital_Output_0 => "DB_Digital_Outputs".Digital_Output_0, Q_Digital_Output_1 => "DB_Digital_Outputs".Digital_Output_1, Q_Digital_Output_2 => "DB_Digital_Outputs".Digital_Output_2, Q_Digital_Output_3 => "DB_Digital_Outputs".Digital_Output_3, Q_Digital_Output_4 => "DB_Digital_Outputs".Digital_Output_4, Q_Digital_Output_5 => "DB_Digital_Outputs".Digital_Output_5, Q_Digital_Output_6 => "DB_Digital_Outputs".Digital_Output_6, Q_Digital_Output_7 => "DB_Digital_Outputs".Digital_Output_7, Q_Digital_Output_8 => "DB_Digital_Outputs".Digital_Output_8, Q_Digital_Output_9 => "DB_Digital_Outputs".Digital_Output_9)
   END_RUNG
   // the same network as SCL:
   "Instance_FB_Digital_Outputs_DB"(DB_Digital_Output_0 := "Digital_Output_0",   // "FB_Digital_Outputs"
                           DB_Digital_Output_1 := "Digital_Output_1",
                           DB_Digital_Output_2 := "Digital_Output_2",
                           DB_Digital_Output_3 := "Digital_Output_3",
                           DB_Digital_Output_4 := "Digital_Output_4",
                           DB_Digital_Output_5 := "Digital_Output_5",
                           DB_Digital_Output_6 := "Digital_Output_6",
                           DB_Digital_Output_7 := "Digital_Output_7",
                           DB_Digital_Output_8 := "Digital_Output_8",
                           DB_Digital_Output_9 := "Digital_Output_9",
                           Q_Digital_Output_0 => "DB_Digital_Outputs".Digital_Output_0,
                           Q_Digital_Output_1 => "DB_Digital_Outputs".Digital_Output_1,
                           Q_Digital_Output_2 => "DB_Digital_Outputs".Digital_Output_2,
                           Q_Digital_Output_3 => "DB_Digital_Outputs".Digital_Output_3,
                           Q_Digital_Output_4 => "DB_Digital_Outputs".Digital_Output_4,
                           Q_Digital_Output_5 => "DB_Digital_Outputs".Digital_Output_5,
                           Q_Digital_Output_6 => "DB_Digital_Outputs".Digital_Output_6,
                           Q_Digital_Output_7 => "DB_Digital_Outputs".Digital_Output_7,
                           Q_Digital_Output_8 => "DB_Digital_Outputs".Digital_Output_8,
                           Q_Digital_Output_9 => "DB_Digital_Outputs".Digital_Output_9);
END_REGION

REGION Network 4
   RUNG wire#powerrail
      "Instance_FB_IO_Device_Functional_Test_DB"(Reset_PLC_Functional_Test := "DB_IO_Device_In_Functional_Test".Reset_PLC_Functional_Test, Status := "DB_IO_Device_In_Functional_Test".Status, Voltage_Read := "Voltage_Read_UInt", Min_Electrical_Current := "DB_Recipe".Min_Electrical_Current, Max_Electrical_Current := "DB_Recipe".Max_Electrical_Current, Time_End_Electrical_Current_Test := "DB_Recipe".Time_End_Electrical_Current_Test, Time_Start_Visual_Test := "DB_Recipe".Time_Start_Visual_Test, In_Functional_Test_Odd := "In_Functional_Test_Odd", In_Functional_Test_Even := "In_Functional_Test_Even", Out_Test_Parameters_Odd => "Out_Test_Parameters_Odd", Out_Test_Parameters_Even => "Out_Test_Parameters_Even", Out_Voltage_Read => "DB_IO_Device_In_Functional_Test".Voltage_Read, Comunication_Error_Panel_1 => "DB_HMI".Alarm_0.%X6, Comunication_Error_Panel_2 => "DB_HMI".Alarm_0.%X7, Comunication_Error_Panel_3 => "DB_HMI".Alarm_0.%X8, Comunication_Error_Panel_4 => "DB_HMI".Alarm_0.%X9, Comunication_Error_Panel_5 => "DB_HMI".Alarm_0.%X10, Comunication_Error_Panel_6 => "DB_HMI".Alarm_0.%X11, Comunication_Error_Panel_7 => "DB_HMI".Alarm_0.%X12, Comunication_Error_Panel_8 => "DB_HMI".Alarm_0.%X13, Comunication_Error_Panel_9 => "DB_HMI".Alarm_0.%X14, Comunication_Error_Panel_10 => "DB_HMI".Alarm_0.%X15, Comunication_Error_Panel_11 => "DB_HMI".Alarm_1.%X0, Comunication_Error_Panel_12 => "DB_HMI".Alarm_1.%X1, Comunication_Error_Panel_13 => "DB_HMI".Alarm_1.%X2, Comunication_Error_Panel_14 => "DB_HMI".Alarm_1.%X3, Comunication_Error_Panel_15 => "DB_HMI".Alarm_1.%X4, Comunication_Error_Panel_16 => "DB_HMI".Alarm_1.%X5, Comunication_Error_Panel_17 => "DB_HMI".Alarm_1.%X6, Comunication_Error_Panel_18 => "DB_HMI".Alarm_1.%X7, Comunication_Error_Panel_19 => "DB_HMI".Alarm_1.%X8, Comunication_Error_Panel_20 => "DB_HMI".Alarm_1.%X9, Comunication_Error_Panel_21 => "DB_HMI".Alarm_1.%X10, Comunication_Error_Panel_22 => "DB_HMI".Alarm_1.%X11, Comunication_Error_Panel_23 => "DB_HMI".Alarm_1.%X12, Comunication_Error_Panel_24 => "DB_HMI".Alarm_1.%X13, Comunication_Error_Panel_25 => "DB_HMI".Alarm_1.%X14, Comunication_Error_Panel_26 => "DB_HMI".Alarm_1.%X15, Comunication_Error_Panel_27 => "DB_HMI".Alarm_2.%X0, Comunication_Error_Panel_28 => "DB_HMI".Alarm_2.%X1, Comunication_Error_Panel_29 => "DB_HMI".Alarm_2.%X2, Comunication_Error_Panel_30 => "DB_HMI".Alarm_2.%X3)
   END_RUNG
   // the same network as SCL:
   "Instance_FB_IO_Device_Functional_Test_DB"(Reset_PLC_Functional_Test := "DB_IO_Device_In_Functional_Test".Reset_PLC_Functional_Test,   // "FB_IO_Device_Functional_Test"
                           Status := "DB_IO_Device_In_Functional_Test".Status,
                           Voltage_Read := "Voltage_Read_UInt",
                           Min_Electrical_Current := "DB_Recipe".Min_Electrical_Current,
                           Max_Electrical_Current := "DB_Recipe".Max_Electrical_Current,
                           Time_End_Electrical_Current_Test := "DB_Recipe".Time_End_Electrical_Current_Test,
                           Time_Start_Visual_Test := "DB_Recipe".Time_Start_Visual_Test,
                           In_Functional_Test_Odd := "In_Functional_Test_Odd",
                           In_Functional_Test_Even := "In_Functional_Test_Even",
                           Out_Test_Parameters_Odd => "Out_Test_Parameters_Odd",
                           Out_Test_Parameters_Even => "Out_Test_Parameters_Even",
                           Out_Voltage_Read => "DB_IO_Device_In_Functional_Test".Voltage_Read,
                           Comunication_Error_Panel_1 => "DB_HMI".Alarm_0.%X6,
                           Comunication_Error_Panel_2 => "DB_HMI".Alarm_0.%X7,
                           Comunication_Error_Panel_3 => "DB_HMI".Alarm_0.%X8,
                           Comunication_Error_Panel_4 => "DB_HMI".Alarm_0.%X9,
                           Comunication_Error_Panel_5 => "DB_HMI".Alarm_0.%X10,
                           Comunication_Error_Panel_6 => "DB_HMI".Alarm_0.%X11,
                           Comunication_Error_Panel_7 => "DB_HMI".Alarm_0.%X12,
                           Comunication_Error_Panel_8 => "DB_HMI".Alarm_0.%X13,
                           Comunication_Error_Panel_9 => "DB_HMI".Alarm_0.%X14,
                           Comunication_Error_Panel_10 => "DB_HMI".Alarm_0.%X15,
                           Comunication_Error_Panel_11 => "DB_HMI".Alarm_1.%X0,
                           Comunication_Error_Panel_12 => "DB_HMI".Alarm_1.%X1,
                           Comunication_Error_Panel_13 => "DB_HMI".Alarm_1.%X2,
                           Comunication_Error_Panel_14 => "DB_HMI".Alarm_1.%X3,
                           Comunication_Error_Panel_15 => "DB_HMI".Alarm_1.%X4,
                           Comunication_Error_Panel_16 => "DB_HMI".Alarm_1.%X5,
                           Comunication_Error_Panel_17 => "DB_HMI".Alarm_1.%X6,
                           Comunication_Error_Panel_18 => "DB_HMI".Alarm_1.%X7,
                           Comunication_Error_Panel_19 => "DB_HMI".Alarm_1.%X8,
                           Comunication_Error_Panel_20 => "DB_HMI".Alarm_1.%X9,
                           Comunication_Error_Panel_21 => "DB_HMI".Alarm_1.%X10,
                           Comunication_Error_Panel_22 => "DB_HMI".Alarm_1.%X11,
                           Comunication_Error_Panel_23 => "DB_HMI".Alarm_1.%X12,
                           Comunication_Error_Panel_24 => "DB_HMI".Alarm_1.%X13,
                           Comunication_Error_Panel_25 => "DB_HMI".Alarm_1.%X14,
                           Comunication_Error_Panel_26 => "DB_HMI".Alarm_1.%X15,
                           Comunication_Error_Panel_27 => "DB_HMI".Alarm_2.%X0,
                           Comunication_Error_Panel_28 => "DB_HMI".Alarm_2.%X1,
                           Comunication_Error_Panel_29 => "DB_HMI".Alarm_2.%X2,
                           Comunication_Error_Panel_30 => "DB_HMI".Alarm_2.%X3);
END_REGION

REGION Network 5
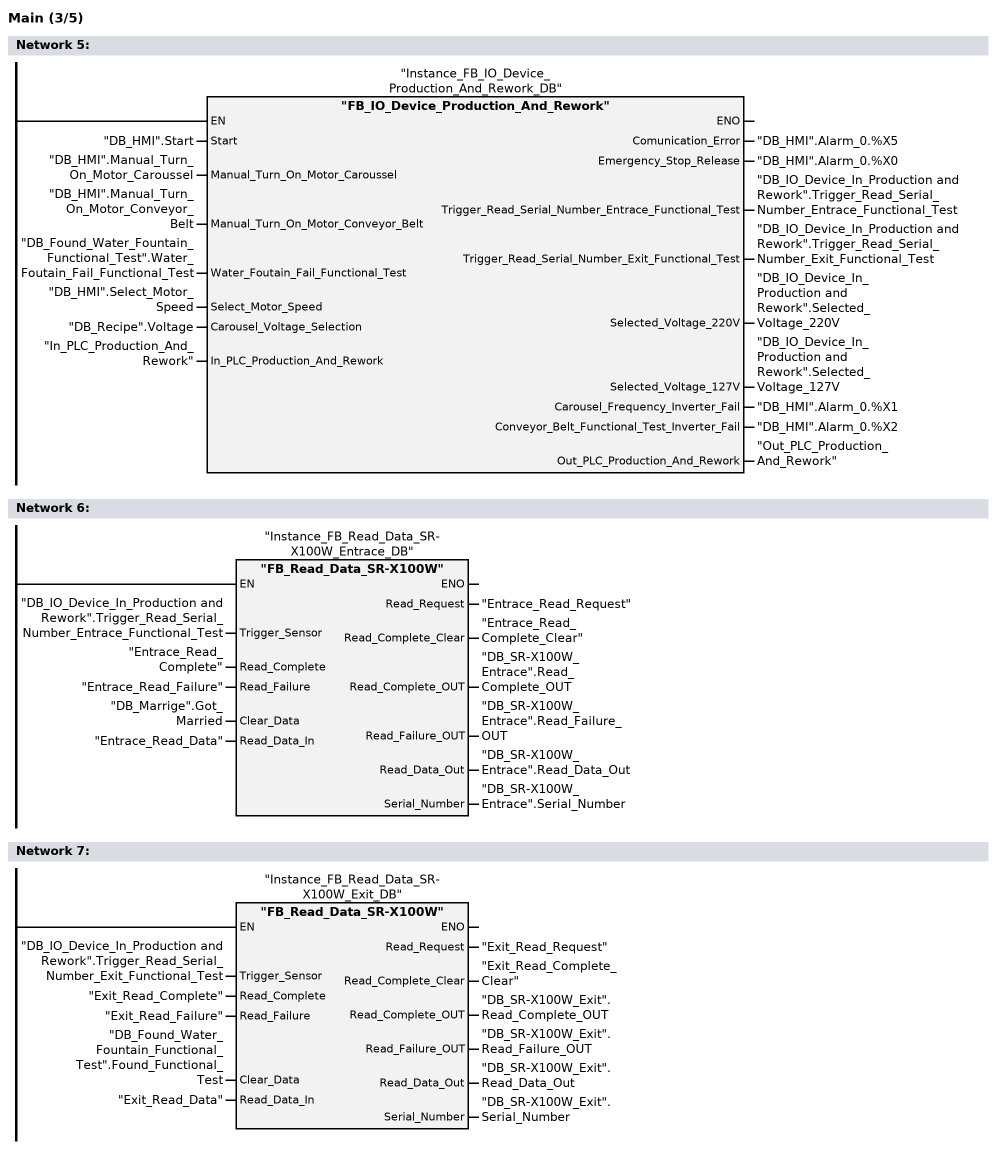
   RUNG wire#powerrail
      "Instance_FB_IO_Device_Production_And_Rework_DB"(Start := "DB_HMI".Start, Manual_Turn_On_Motor_Caroussel := "DB_HMI".Manual_Turn_On_Motor_Caroussel, Manual_Turn_On_Motor_Conveyor_Belt := "DB_HMI".Manual_Turn_On_Motor_Conveyor_Belt, Water_Foutain_Fail_Functional_Test := "DB_Found_Water_Fountain_Functional_Test".Water_Foutain_Fail_Functional_Test, Select_Motor_Speed := "DB_HMI".Select_Motor_Speed, Carousel_Voltage_Selection := "DB_Recipe".Voltage, In_PLC_Production_And_Rework := "In_PLC_Production_And_Rework", Comunication_Error => "DB_HMI".Alarm_0.%X5, Emergency_Stop_Release => "DB_HMI".Alarm_0.%X0, Trigger_Read_Serial_Number_Entrace_Functional_Test => "DB_IO_Device_In_Production and Rework".Trigger_Read_Serial_Number_Entrace_Functional_Test, Trigger_Read_Serial_Number_Exit_Functional_Test => "DB_IO_Device_In_Production and Rework".Trigger_Read_Serial_Number_Exit_Functional_Test, Selected_Voltage_220V => "DB_IO_Device_In_Production and Rework".Selected_Voltage_220V, Selected_Voltage_127V => "DB_IO_Device_In_Production and Rework".Selected_Voltage_127V, Carousel_Frequency_Inverter_Fail => "DB_HMI".Alarm_0.%X1, Conveyor_Belt_Functional_Test_Inverter_Fail => "DB_HMI".Alarm_0.%X2, Out_PLC_Production_And_Rework => "Out_PLC_Production_And_Rework")
   END_RUNG
   // the same network as SCL:
   "Instance_FB_IO_Device_Production_And_Rework_DB"(Start := "DB_HMI".Start,   // "FB_IO_Device_Production_And_Rework"
                           Manual_Turn_On_Motor_Caroussel := "DB_HMI".Manual_Turn_On_Motor_Caroussel,
                           Manual_Turn_On_Motor_Conveyor_Belt := "DB_HMI".Manual_Turn_On_Motor_Conveyor_Belt,
                           Water_Foutain_Fail_Functional_Test := "DB_Found_Water_Fountain_Functional_Test".Water_Foutain_Fail_Functional_Test,
                           Select_Motor_Speed := "DB_HMI".Select_Motor_Speed,
                           Carousel_Voltage_Selection := "DB_Recipe".Voltage,
                           In_PLC_Production_And_Rework := "In_PLC_Production_And_Rework",
                           Comunication_Error => "DB_HMI".Alarm_0.%X5,
                           Emergency_Stop_Release => "DB_HMI".Alarm_0.%X0,
                           Trigger_Read_Serial_Number_Entrace_Functional_Test => "DB_IO_Device_In_Production and Rework".Trigger_Read_Serial_Number_Entrace_Functional_Test,
                           Trigger_Read_Serial_Number_Exit_Functional_Test => "DB_IO_Device_In_Production and Rework".Trigger_Read_Serial_Number_Exit_Functional_Test,
                           Selected_Voltage_220V => "DB_IO_Device_In_Production and Rework".Selected_Voltage_220V,
                           Selected_Voltage_127V => "DB_IO_Device_In_Production and Rework".Selected_Voltage_127V,
                           Carousel_Frequency_Inverter_Fail => "DB_HMI".Alarm_0.%X1,
                           Conveyor_Belt_Functional_Test_Inverter_Fail => "DB_HMI".Alarm_0.%X2,
                           Out_PLC_Production_And_Rework => "Out_PLC_Production_And_Rework");
END_REGION

REGION Network 6
   RUNG wire#powerrail
      "Instance_FB_Read_Data_SR-X100W_Entrace_DB"(Trigger_Sensor := "DB_IO_Device_In_Production and Rework".Trigger_Read_Serial_Number_Entrace_Functional_Test, Read_Complete := "Entrace_Read_Complete", Read_Failure := "Entrace_Read_Failure", Clear_Data := "DB_Marrige".Got_Married, Read_Data_In := "Entrace_Read_Data", Read_Request => "Entrace_Read_Request", Read_Complete_Clear => "Entrace_Read_Complete_Clear", Read_Complete_OUT => "DB_SR-X100W_Entrace".Read_Complete_OUT, Read_Failure_OUT => "DB_SR-X100W_Entrace".Read_Failure_OUT, Read_Data_Out => "DB_SR-X100W_Entrace".Read_Data_Out, Serial_Number => "DB_SR-X100W_Entrace".Serial_Number)
   END_RUNG
   // the same network as SCL:
   "Instance_FB_Read_Data_SR-X100W_Entrace_DB"(Trigger_Sensor := "DB_IO_Device_In_Production and Rework".Trigger_Read_Serial_Number_Entrace_Functional_Test,   // "FB_Read_Data_SR-X100W"
                           Read_Complete := "Entrace_Read_Complete",
                           Read_Failure := "Entrace_Read_Failure",
                           Clear_Data := "DB_Marrige".Got_Married,
                           Read_Data_In := "Entrace_Read_Data",
                           Read_Request => "Entrace_Read_Request",
                           Read_Complete_Clear => "Entrace_Read_Complete_Clear",
                           Read_Complete_OUT => "DB_SR-X100W_Entrace".Read_Complete_OUT,
                           Read_Failure_OUT => "DB_SR-X100W_Entrace".Read_Failure_OUT,
                           Read_Data_Out => "DB_SR-X100W_Entrace".Read_Data_Out,
                           Serial_Number => "DB_SR-X100W_Entrace".Serial_Number);
END_REGION

REGION Network 7
   RUNG wire#powerrail
      "Instance_FB_Read_Data_SR-X100W_Exit_DB"(Trigger_Sensor := "DB_IO_Device_In_Production and Rework".Trigger_Read_Serial_Number_Exit_Functional_Test, Read_Complete := "Exit_Read_Complete", Read_Failure := "Exit_Read_Failure", Clear_Data := "DB_Found_Water_Fountain_Functional_Test".Found_Functional_Test, Read_Data_In := "Exit_Read_Data", Read_Request => "Exit_Read_Request", Read_Complete_Clear => "Exit_Read_Complete_Clear", Read_Complete_OUT => "DB_SR-X100W_Exit".Read_Complete_OUT, Read_Failure_OUT => "DB_SR-X100W_Exit".Read_Failure_OUT, Read_Data_Out => "DB_SR-X100W_Exit".Read_Data_Out, Serial_Number => "DB_SR-X100W_Exit".Serial_Number)
   END_RUNG
   // the same network as SCL:
   "Instance_FB_Read_Data_SR-X100W_Exit_DB"(Trigger_Sensor := "DB_IO_Device_In_Production and Rework".Trigger_Read_Serial_Number_Exit_Functional_Test,   // "FB_Read_Data_SR-X100W"
                           Read_Complete := "Exit_Read_Complete",
                           Read_Failure := "Exit_Read_Failure",
                           Clear_Data := "DB_Found_Water_Fountain_Functional_Test".Found_Functional_Test,
                           Read_Data_In := "Exit_Read_Data",
                           Read_Request => "Exit_Read_Request",
                           Read_Complete_Clear => "Exit_Read_Complete_Clear",
                           Read_Complete_OUT => "DB_SR-X100W_Exit".Read_Complete_OUT,
                           Read_Failure_OUT => "DB_SR-X100W_Exit".Read_Failure_OUT,
                           Read_Data_Out => "DB_SR-X100W_Exit".Read_Data_Out,
                           Serial_Number => "DB_SR-X100W_Exit".Serial_Number);
END_REGION

REGION Network 8
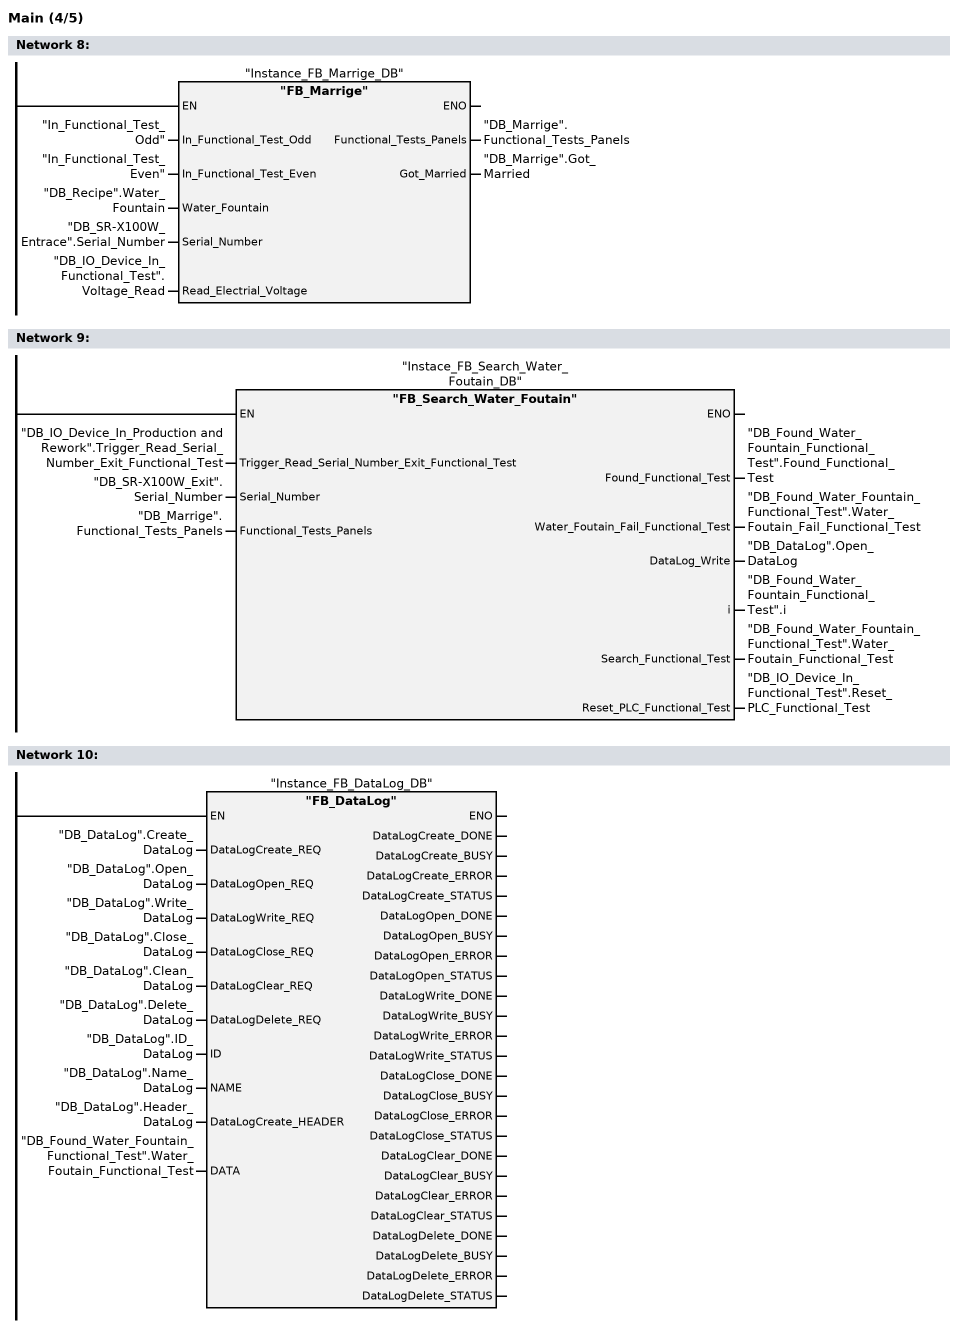
   RUNG wire#powerrail
      "Instance_FB_Marrige_DB"(In_Functional_Test_Odd := "In_Functional_Test_Odd", In_Functional_Test_Even := "In_Functional_Test_Even", Water_Fountain := "DB_Recipe".Water_Fountain, Serial_Number := "DB_SR-X100W_Entrace".Serial_Number, Read_Electrial_Voltage := "DB_IO_Device_In_Functional_Test".Voltage_Read, Functional_Tests_Panels => "DB_Marrige".Functional_Tests_Panels, Got_Married => "DB_Marrige".Got_Married)
   END_RUNG
   // the same network as SCL:
   "Instance_FB_Marrige_DB"(In_Functional_Test_Odd := "In_Functional_Test_Odd",   // "FB_Marrige"
                           In_Functional_Test_Even := "In_Functional_Test_Even",
                           Water_Fountain := "DB_Recipe".Water_Fountain,
                           Serial_Number := "DB_SR-X100W_Entrace".Serial_Number,
                           Read_Electrial_Voltage := "DB_IO_Device_In_Functional_Test".Voltage_Read,
                           Functional_Tests_Panels => "DB_Marrige".Functional_Tests_Panels,
                           Got_Married => "DB_Marrige".Got_Married);
END_REGION

REGION Network 9
   RUNG wire#powerrail
      "Instace_FB_Search_Water_Foutain_DB"(Trigger_Read_Serial_Number_Exit_Functional_Test := "DB_IO_Device_In_Production and Rework".Trigger_Read_Serial_Number_Exit_Functional_Test, Serial_Number := "DB_SR-X100W_Exit".Serial_Number, Functional_Tests_Panels := "DB_Marrige".Functional_Tests_Panels, Found_Functional_Test => "DB_Found_Water_Fountain_Functional_Test".Found_Functional_Test, Water_Foutain_Fail_Functional_Test => "DB_Found_Water_Fountain_Functional_Test".Water_Foutain_Fail_Functional_Test, DataLog_Write => "DB_DataLog".Open_DataLog, i => "DB_Found_Water_Fountain_Functional_Test".i, Search_Functional_Test => "DB_Found_Water_Fountain_Functional_Test".Water_Foutain_Functional_Test, Reset_PLC_Functional_Test => "DB_IO_Device_In_Functional_Test".Reset_PLC_Functional_Test)
   END_RUNG
   // the same network as SCL:
   "Instace_FB_Search_Water_Foutain_DB"(Trigger_Read_Serial_Number_Exit_Functional_Test := "DB_IO_Device_In_Production and Rework".Trigger_Read_Serial_Number_Exit_Functional_Test,   // "FB_Search_Water_Foutain"
                           Serial_Number := "DB_SR-X100W_Exit".Serial_Number,
                           Functional_Tests_Panels := "DB_Marrige".Functional_Tests_Panels,
                           Found_Functional_Test => "DB_Found_Water_Fountain_Functional_Test".Found_Functional_Test,
                           Water_Foutain_Fail_Functional_Test => "DB_Found_Water_Fountain_Functional_Test".Water_Foutain_Fail_Functional_Test,
                           DataLog_Write => "DB_DataLog".Open_DataLog,
                           i => "DB_Found_Water_Fountain_Functional_Test".i,
                           Search_Functional_Test => "DB_Found_Water_Fountain_Functional_Test".Water_Foutain_Functional_Test,
                           Reset_PLC_Functional_Test => "DB_IO_Device_In_Functional_Test".Reset_PLC_Functional_Test);
END_REGION

REGION Network 10
   RUNG wire#powerrail
      "Instance_FB_DataLog_DB"(DataLogCreate_REQ := "DB_DataLog".Create_DataLog, DataLogOpen_REQ := "DB_DataLog".Open_DataLog, DataLogWrite_REQ := "DB_DataLog".Write_DataLog, DataLogClose_REQ := "DB_DataLog".Close_DataLog, DataLogClear_REQ := "DB_DataLog".Clean_DataLog, DataLogDelete_REQ := "DB_DataLog".Delete_DataLog, ID := "DB_DataLog".ID_DataLog, "NAME" := "DB_DataLog".Name_DataLog, DataLogCreate_HEADER := "DB_DataLog".Header_DataLog, DATA := "DB_Found_Water_Fountain_Functional_Test".Water_Foutain_Functional_Test, DataLogCreate_DONE =>, DataLogCreate_BUSY =>, DataLogCreate_ERROR =>, DataLogCreate_STATUS =>, DataLogOpen_DONE =>, DataLogOpen_BUSY =>, DataLogOpen_ERROR =>, DataLogOpen_STATUS =>, DataLogWrite_DONE =>, DataLogWrite_BUSY =>, DataLogWrite_ERROR =>, DataLogWrite_STATUS =>, DataLogClose_DONE =>, DataLogClose_BUSY =>, DataLogClose_ERROR =>, DataLogClose_STATUS =>, DataLogClear_DONE =>, DataLogClear_BUSY =>, DataLogClear_ERROR =>, DataLogClear_STATUS =>, DataLogDelete_DONE =>, DataLogDelete_BUSY =>, DataLogDelete_ERROR =>, DataLogDelete_STATUS =>)
   END_RUNG
   // the same network as SCL:
   "Instance_FB_DataLog_DB"(DataLogCreate_REQ := "DB_DataLog".Create_DataLog,   // "FB_DataLog"
                           DataLogOpen_REQ := "DB_DataLog".Open_DataLog,
                           DataLogWrite_REQ := "DB_DataLog".Write_DataLog,
                           DataLogClose_REQ := "DB_DataLog".Close_DataLog,
                           DataLogClear_REQ := "DB_DataLog".Clean_DataLog,
                           DataLogDelete_REQ := "DB_DataLog".Delete_DataLog,
                           ID := "DB_DataLog".ID_DataLog,
                           "NAME" := "DB_DataLog".Name_DataLog,
                           DataLogCreate_HEADER := "DB_DataLog".Header_DataLog,
                           DATA := "DB_Found_Water_Fountain_Functional_Test".Water_Foutain_Functional_Test);
END_REGION

REGION Network 11
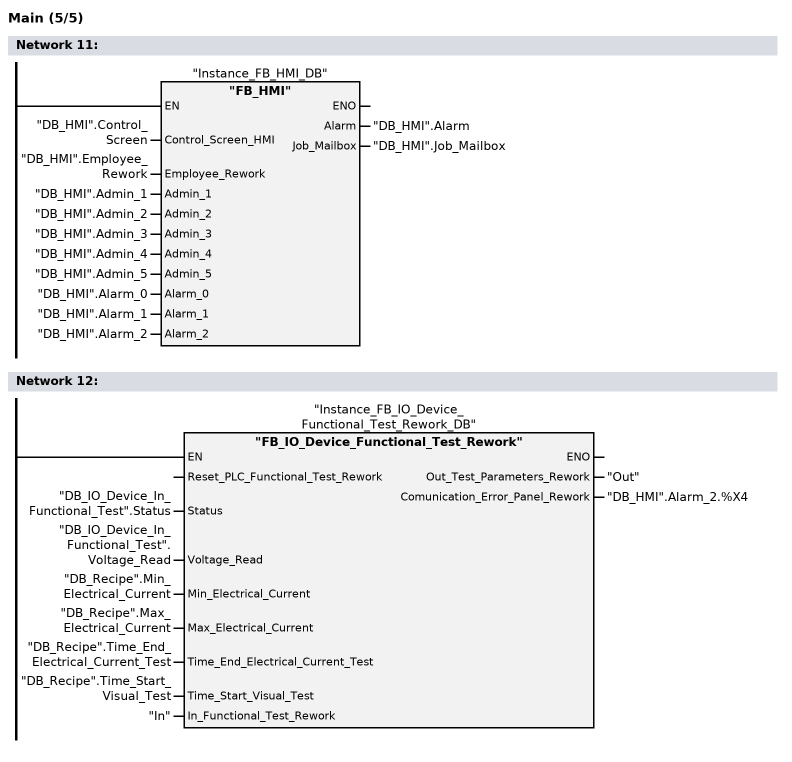
   RUNG wire#powerrail
      "Instance_FB_HMI_DB"(Control_Screen_HMI := "DB_HMI".Control_Screen, Employee_Rework := "DB_HMI".Employee_Rework, Admin_1 := "DB_HMI".Admin_1, Admin_2 := "DB_HMI".Admin_2, Admin_3 := "DB_HMI".Admin_3, Admin_4 := "DB_HMI".Admin_4, Admin_5 := "DB_HMI".Admin_5, Alarm_0 := "DB_HMI".Alarm_0, Alarm_1 := "DB_HMI".Alarm_1, Alarm_2 := "DB_HMI".Alarm_2, Alarm => "DB_HMI".Alarm, Job_Mailbox => "DB_HMI".Job_Mailbox)
   END_RUNG
   // the same network as SCL:
   "Instance_FB_HMI_DB"(Control_Screen_HMI := "DB_HMI".Control_Screen,   // "FB_HMI"
                        Employee_Rework := "DB_HMI".Employee_Rework,
                        Admin_1 := "DB_HMI".Admin_1,
                        Admin_2 := "DB_HMI".Admin_2,
                        Admin_3 := "DB_HMI".Admin_3,
                        Admin_4 := "DB_HMI".Admin_4,
                        Admin_5 := "DB_HMI".Admin_5,
                        Alarm_0 := "DB_HMI".Alarm_0,
                        Alarm_1 := "DB_HMI".Alarm_1,
                        Alarm_2 := "DB_HMI".Alarm_2,
                        Alarm => "DB_HMI".Alarm,
                        Job_Mailbox => "DB_HMI".Job_Mailbox);
END_REGION

REGION Network 12
   RUNG wire#powerrail
      "Instance_FB_IO_Device_Functional_Test_Rework_DB"(Reset_PLC_Functional_Test_Rework :=, Status := "DB_IO_Device_In_Functional_Test".Status, Voltage_Read := "DB_IO_Device_In_Functional_Test".Voltage_Read, Min_Electrical_Current := "DB_Recipe".Min_Electrical_Current, Max_Electrical_Current := "DB_Recipe".Max_Electrical_Current, Time_End_Electrical_Current_Test := "DB_Recipe".Time_End_Electrical_Current_Test, Time_Start_Visual_Test := "DB_Recipe".Time_Start_Visual_Test, In_Functional_Test_Rework := "In", Out_Test_Parameters_Rework => "Out", Comunication_Error_Panel_Rework => "DB_HMI".Alarm_2.%X4)
   END_RUNG
   // the same network as SCL:
   "Instance_FB_IO_Device_Functional_Test_Rework_DB"(Status := "DB_IO_Device_In_Functional_Test".Status,   // "FB_IO_Device_Functional_Test_Rework"
                           Voltage_Read := "DB_IO_Device_In_Functional_Test".Voltage_Read,
                           Min_Electrical_Current := "DB_Recipe".Min_Electrical_Current,
                           Max_Electrical_Current := "DB_Recipe".Max_Electrical_Current,
                           Time_End_Electrical_Current_Test := "DB_Recipe".Time_End_Electrical_Current_Test,
                           Time_Start_Visual_Test := "DB_Recipe".Time_Start_Visual_Test,
                           In_Functional_Test_Rework := "In",
                           Out_Test_Parameters_Rework => "Out",
                           Comunication_Error_Panel_Rework => "DB_HMI".Alarm_2.%X4);
END_REGION
END_ORGANIZATION_BLOCK

FUNCTION_BLOCK "FB_Digita_Inputs"   // FB1, LAD
{ S7_Optimized_Access := 'TRUE' }
// stored: MemoryReserve 100, SetENOAutomatically false
   VAR_INPUT
      "I-Digital_Input_0" : Bool;
      "I-Digital_Input_1" : Bool;
      "I-Digital_Input_2" : Bool;
      "I-Digital_Input_3" : Bool;
      "I-Digital_Input_4" : Bool;
      "I-Digital_Input_5" : Bool;
      "I-Digital_Input_6" : Bool;
      "I-Digital_Input_7" : Bool;
      "I-Digital_Input_8" : Bool;
      "I-Digital_Input_9" : Bool;
      "I-Digital_Input_10" : Bool;
      "I-Digital_Input_11" : Bool;
      "I-Digital_Input_12" : Bool;
      "I-Digital_Input_13" : Bool;
   END_VAR
   VAR_OUTPUT
      DB_Digital_Input_0 : Bool;
      DB_Digital_Input_1 : Bool;
      DB_Digital_Input_2 : Bool;
      DB_Digital_Input_3 : Bool;
      DB_Digital_Input_4 : Bool;
      DB_Digital_Input_5 : Bool;
      DB_Digital_Input_6 : Bool;
      DB_Digital_Input_7 : Bool;
      DB_Digital_Input_8 : Bool;
      DB_Digital_Input_9 : Bool;
      DB_Digital_Input_10 : Bool;
      DB_Digital_Input_11 : Bool;
      DB_Digital_Input_12 : Bool;
      DB_Digital_Input_13 : Bool;
   END_VAR
BEGIN

REGION Network 1
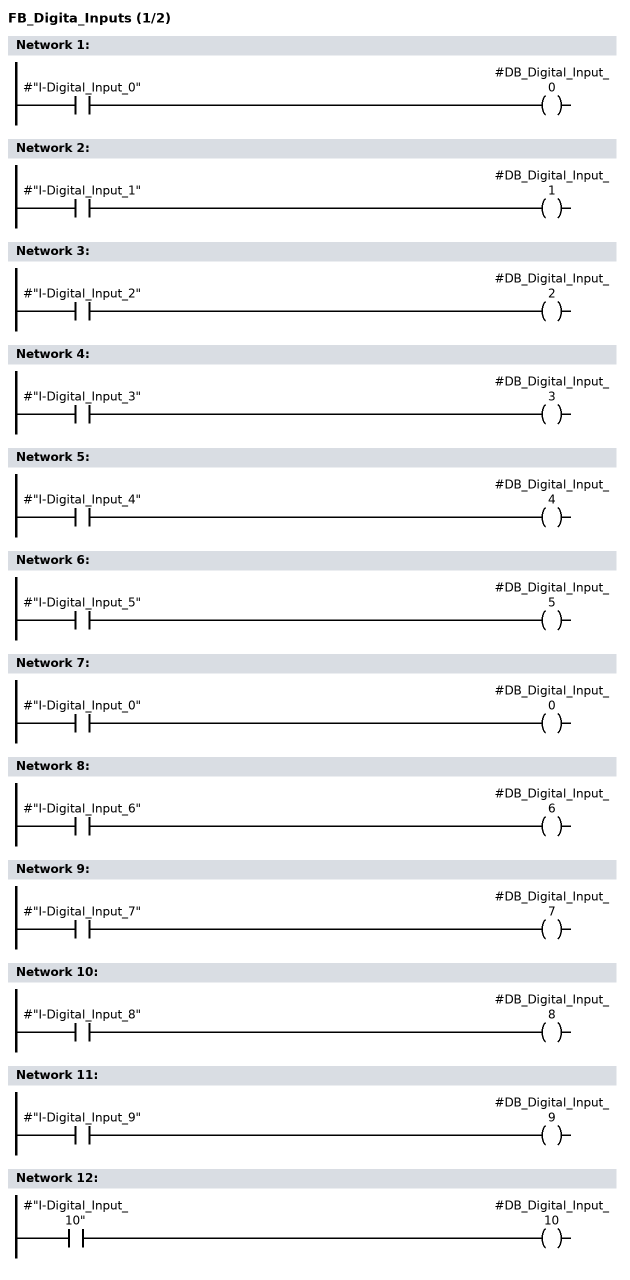
   RUNG wire#powerrail
      Contact( #"I-Digital_Input_0" )
      Coil( #DB_Digital_Input_0 )
   END_RUNG
   // the same network as SCL:
   #DB_Digital_Input_0 := #"I-Digital_Input_0";
END_REGION

REGION Network 2
   RUNG wire#powerrail
      Contact( #"I-Digital_Input_1" )
      Coil( #DB_Digital_Input_1 )
   END_RUNG
   // the same network as SCL:
   #DB_Digital_Input_1 := #"I-Digital_Input_1";
END_REGION

REGION Network 3
   RUNG wire#powerrail
      Contact( #"I-Digital_Input_2" )
      Coil( #DB_Digital_Input_2 )
   END_RUNG
   // the same network as SCL:
   #DB_Digital_Input_2 := #"I-Digital_Input_2";
END_REGION

REGION Network 4
   RUNG wire#powerrail
      Contact( #"I-Digital_Input_3" )
      Coil( #DB_Digital_Input_3 )
   END_RUNG
   // the same network as SCL:
   #DB_Digital_Input_3 := #"I-Digital_Input_3";
END_REGION

REGION Network 5
   RUNG wire#powerrail
      Contact( #"I-Digital_Input_4" )
      Coil( #DB_Digital_Input_4 )
   END_RUNG
   // the same network as SCL:
   #DB_Digital_Input_4 := #"I-Digital_Input_4";
END_REGION

REGION Network 6
   RUNG wire#powerrail
      Contact( #"I-Digital_Input_5" )
      Coil( #DB_Digital_Input_5 )
   END_RUNG
   // the same network as SCL:
   #DB_Digital_Input_5 := #"I-Digital_Input_5";
END_REGION

REGION Network 7
   RUNG wire#powerrail
      Contact( #"I-Digital_Input_0" )
      Coil( #DB_Digital_Input_0 )
   END_RUNG
   // the same network as SCL:
   #DB_Digital_Input_0 := #"I-Digital_Input_0";
END_REGION

REGION Network 8
   RUNG wire#powerrail
      Contact( #"I-Digital_Input_6" )
      Coil( #DB_Digital_Input_6 )
   END_RUNG
   // the same network as SCL:
   #DB_Digital_Input_6 := #"I-Digital_Input_6";
END_REGION

REGION Network 9
   RUNG wire#powerrail
      Contact( #"I-Digital_Input_7" )
      Coil( #DB_Digital_Input_7 )
   END_RUNG
   // the same network as SCL:
   #DB_Digital_Input_7 := #"I-Digital_Input_7";
END_REGION

REGION Network 10
   RUNG wire#powerrail
      Contact( #"I-Digital_Input_8" )
      Coil( #DB_Digital_Input_8 )
   END_RUNG
   // the same network as SCL:
   #DB_Digital_Input_8 := #"I-Digital_Input_8";
END_REGION

REGION Network 11
   RUNG wire#powerrail
      Contact( #"I-Digital_Input_9" )
      Coil( #DB_Digital_Input_9 )
   END_RUNG
   // the same network as SCL:
   #DB_Digital_Input_9 := #"I-Digital_Input_9";
END_REGION

REGION Network 12
   RUNG wire#powerrail
      Contact( #"I-Digital_Input_10" )
      Coil( #DB_Digital_Input_10 )
   END_RUNG
   // the same network as SCL:
   #DB_Digital_Input_10 := #"I-Digital_Input_10";
END_REGION

REGION Network 13
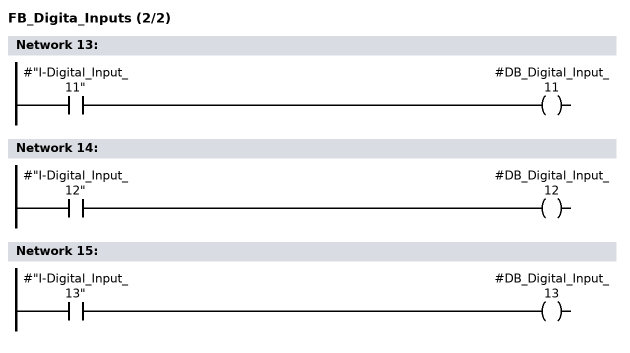
   RUNG wire#powerrail
      Contact( #"I-Digital_Input_11" )
      Coil( #DB_Digital_Input_11 )
   END_RUNG
   // the same network as SCL:
   #DB_Digital_Input_11 := #"I-Digital_Input_11";
END_REGION

REGION Network 14
   RUNG wire#powerrail
      Contact( #"I-Digital_Input_12" )
      Coil( #DB_Digital_Input_12 )
   END_RUNG
   // the same network as SCL:
   #DB_Digital_Input_12 := #"I-Digital_Input_12";
END_REGION

REGION Network 15
   RUNG wire#powerrail
      Contact( #"I-Digital_Input_13" )
      Coil( #DB_Digital_Input_13 )
   END_RUNG
   // the same network as SCL:
   #DB_Digital_Input_13 := #"I-Digital_Input_13";
END_REGION
END_FUNCTION_BLOCK

FUNCTION_BLOCK "FB_Digital_Outputs"   // FB3, LAD
{ S7_Optimized_Access := 'TRUE' }
// stored: MemoryReserve 100, SetENOAutomatically false
   VAR_INPUT
      DB_Digital_Output_0 : Bool;
      DB_Digital_Output_1 : Bool;
      DB_Digital_Output_2 : Bool;
      DB_Digital_Output_3 : Bool;
      DB_Digital_Output_4 : Bool;
      DB_Digital_Output_5 : Bool;
      DB_Digital_Output_6 : Bool;
      DB_Digital_Output_7 : Bool;
      DB_Digital_Output_8 : Bool;
      DB_Digital_Output_9 : Bool;
   END_VAR
   VAR_OUTPUT
      Q_Digital_Output_0 : Bool;
      Q_Digital_Output_1 : Bool;
      Q_Digital_Output_2 : Bool;
      Q_Digital_Output_3 : Bool;
      Q_Digital_Output_4 : Bool;
      Q_Digital_Output_5 : Bool;
      Q_Digital_Output_6 : Bool;
      Q_Digital_Output_7 : Bool;
      Q_Digital_Output_8 : Bool;
      Q_Digital_Output_9 : Bool;
   END_VAR
BEGIN

REGION Network 1
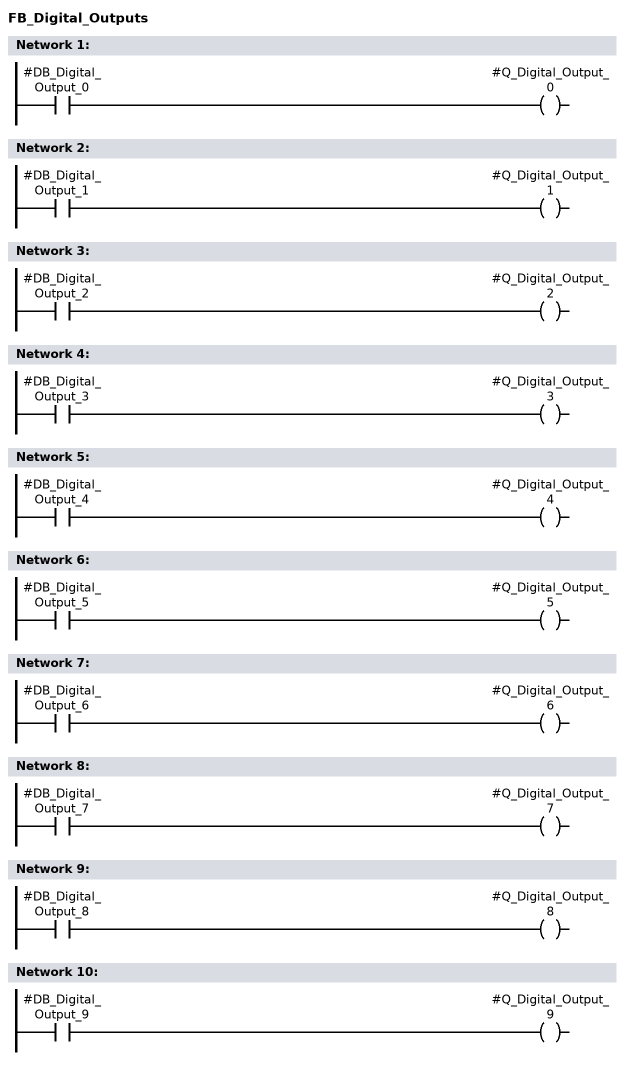
   RUNG wire#powerrail
      Contact( #DB_Digital_Output_0 )
      Coil( #Q_Digital_Output_0 )
   END_RUNG
   // the same network as SCL:
   #Q_Digital_Output_0 := #DB_Digital_Output_0;
END_REGION

REGION Network 2
   RUNG wire#powerrail
      Contact( #DB_Digital_Output_1 )
      Coil( #Q_Digital_Output_1 )
   END_RUNG
   // the same network as SCL:
   #Q_Digital_Output_1 := #DB_Digital_Output_1;
END_REGION

REGION Network 3
   RUNG wire#powerrail
      Contact( #DB_Digital_Output_2 )
      Coil( #Q_Digital_Output_2 )
   END_RUNG
   // the same network as SCL:
   #Q_Digital_Output_2 := #DB_Digital_Output_2;
END_REGION

REGION Network 4
   RUNG wire#powerrail
      Contact( #DB_Digital_Output_3 )
      Coil( #Q_Digital_Output_3 )
   END_RUNG
   // the same network as SCL:
   #Q_Digital_Output_3 := #DB_Digital_Output_3;
END_REGION

REGION Network 5
   RUNG wire#powerrail
      Contact( #DB_Digital_Output_4 )
      Coil( #Q_Digital_Output_4 )
   END_RUNG
   // the same network as SCL:
   #Q_Digital_Output_4 := #DB_Digital_Output_4;
END_REGION

REGION Network 6
   RUNG wire#powerrail
      Contact( #DB_Digital_Output_5 )
      Coil( #Q_Digital_Output_5 )
   END_RUNG
   // the same network as SCL:
   #Q_Digital_Output_5 := #DB_Digital_Output_5;
END_REGION

REGION Network 7
   RUNG wire#powerrail
      Contact( #DB_Digital_Output_6 )
      Coil( #Q_Digital_Output_6 )
   END_RUNG
   // the same network as SCL:
   #Q_Digital_Output_6 := #DB_Digital_Output_6;
END_REGION

REGION Network 8
   RUNG wire#powerrail
      Contact( #DB_Digital_Output_7 )
      Coil( #Q_Digital_Output_7 )
   END_RUNG
   // the same network as SCL:
   #Q_Digital_Output_7 := #DB_Digital_Output_7;
END_REGION

REGION Network 9
   RUNG wire#powerrail
      Contact( #DB_Digital_Output_8 )
      Coil( #Q_Digital_Output_8 )
   END_RUNG
   // the same network as SCL:
   #Q_Digital_Output_8 := #DB_Digital_Output_8;
END_REGION

REGION Network 10
   RUNG wire#powerrail
      Contact( #DB_Digital_Output_9 )
      Coil( #Q_Digital_Output_9 )
   END_RUNG
   // the same network as SCL:
   #Q_Digital_Output_9 := #DB_Digital_Output_9;
END_REGION
END_FUNCTION_BLOCK

FUNCTION_BLOCK "FB_IO_Device_Functional_Test"   // FB4, LAD
{ S7_Optimized_Access := 'TRUE' }
// stored: MemoryReserve 100, SetENOAutomatically false
   VAR_INPUT
      Reset_PLC_Functional_Test : Array[0..31] of Bool;
      Status : Bool;
      Voltage_Read : UInt;
      Min_Electrical_Current : UInt;
      Max_Electrical_Current : UInt;
      Time_End_Electrical_Current_Test : Time;
      Time_Start_Visual_Test : Time;
      In_Functional_Test_Odd : "IO_Device_Functinal_Test_Odd";
      In_Functional_Test_Even : "IO_Device_Functinal_Test_Even";
   END_VAR
   VAR_OUTPUT
      Out_Test_Parameters_Odd : "IO_Device_Test_Parameters_Odd";
      Out_Test_Parameters_Even : "IO_Device_Test_Parameters_Even";
      Out_Voltage_Read : UInt;
      Comunication_Error_Panel_1 : Bool;
      Comunication_Error_Panel_2 : Bool;
      Comunication_Error_Panel_3 : Bool;
      Comunication_Error_Panel_4 : Bool;
      Comunication_Error_Panel_5 : Bool;
      Comunication_Error_Panel_6 : Bool;
      Comunication_Error_Panel_7 : Bool;
      Comunication_Error_Panel_8 : Bool;
      Comunication_Error_Panel_9 : Bool;
      Comunication_Error_Panel_10 : Bool;
      Comunication_Error_Panel_11 : Bool;
      Comunication_Error_Panel_12 : Bool;
      Comunication_Error_Panel_13 : Bool;
      Comunication_Error_Panel_14 : Bool;
      Comunication_Error_Panel_15 : Bool;
      Comunication_Error_Panel_16 : Bool;
      Comunication_Error_Panel_17 : Bool;
      Comunication_Error_Panel_18 : Bool;
      Comunication_Error_Panel_19 : Bool;
      Comunication_Error_Panel_20 : Bool;
      Comunication_Error_Panel_21 : Bool;
      Comunication_Error_Panel_22 : Bool;
      Comunication_Error_Panel_23 : Bool;
      Comunication_Error_Panel_24 : Bool;
      Comunication_Error_Panel_25 : Bool;
      Comunication_Error_Panel_26 : Bool;
      Comunication_Error_Panel_27 : Bool;
      Comunication_Error_Panel_28 : Bool;
      Comunication_Error_Panel_29 : Bool;
      Comunication_Error_Panel_30 : Bool;
   END_VAR
   VAR
      Enable_Comunication_Erro_3 : Bool;
      Enable_Comunication_Erro_4 : Bool;
      Enable_Comunication_Erro_5 : Bool;
      Enable_Comunication_Erro_6 : Bool;
      Enable_Comunication_Erro_7 : Bool;
      Enable_Comunication_Erro_8 : Bool;
      Enable_Comunication_Erro_9 : Bool;
      Enable_Comunication_Erro_10 : Bool;
      Enable_Comunication_Erro_11 : Bool;
      Enable_Comunication_Erro_12 : Bool;
      Enable_Comunication_Erro_13 : Bool;
      Enable_Comunication_Erro_14 : Bool;
      Enable_Comunication_Erro_15 : Bool;
      Enable_Comunication_Erro_16 : Bool;
      Enable_Comunication_Erro_17 : Bool;
      Enable_Comunication_Erro_18 : Bool;
      Enable_Comunication_Erro_19 : Bool;
      Enable_Comunication_Erro_20 : Bool;
      Enable_Comunication_Erro_21 : Bool;
      Enable_Comunication_Erro_22 : Bool;
      Enable_Comunication_Erro_23 : Bool;
      Enable_Comunication_Erro_24 : Bool;
      Enable_Comunication_Erro_25 : Bool;
      Enable_Comunication_Erro_26 : Bool;
      Enable_Comunication_Erro_27 : Bool;
      Enable_Comunication_Erro_28 : Bool;
      Enable_Comunication_Erro_29 : Bool;
      Enable_Comunication_Erro_30 : Bool;
      Timer_Alarme_A_1 { S7_SetPoint := 'True'} : TON_TIME;
      Timer_Alarme_B_1 { S7_SetPoint := 'True'} : TON_TIME;
      Timer_Alarme_A_2 { S7_SetPoint := 'True'} : TON_TIME;
      Timer_Alarme_B_2 { S7_SetPoint := 'True'} : TON_TIME;
      Timer_Alarme_A_3 { S7_SetPoint := 'True'} : TON_TIME;
      Timer_Alarme_B_3 { S7_SetPoint := 'True'} : TON_TIME;
      Timer_Alarme_A_4 { S7_SetPoint := 'True'} : TON_TIME;
      Timer_Alarme_B_4 { S7_SetPoint := 'True'} : TON_TIME;
      Timer_Alarme_A_5 { S7_SetPoint := 'True'} : TON_TIME;
      Timer_Alarme_B_5 { S7_SetPoint := 'True'} : TON_TIME;
      Timer_Alarme_A_6 { S7_SetPoint := 'True'} : TON_TIME;
      Timer_Alarme_B_6 { S7_SetPoint := 'True'} : TON_TIME;
      Timer_Alarme_A_7 { S7_SetPoint := 'True'} : TON_TIME;
      Timer_Alarme_B_7 { S7_SetPoint := 'True'} : TON_TIME;
      Timer_Alarme_A_8 { S7_SetPoint := 'True'} : TON_TIME;
      Timer_Alarme_B_8 { S7_SetPoint := 'True'} : TON_TIME;
      Timer_Alarme_A_9 { S7_SetPoint := 'True'} : TON_TIME;
      Timer_Alarme_B_9 { S7_SetPoint := 'True'} : TON_TIME;
      Timer_Alarme_A_10 { S7_SetPoint := 'True'} : TON_TIME;
      Timer_Alarme_B_10 { S7_SetPoint := 'True'} : TON_TIME;
      Timer_Alarme_A_11 { S7_SetPoint := 'True'} : TON_TIME;
      Timer_Alarme_B_11 { S7_SetPoint := 'True'} : TON_TIME;
      Timer_Alarme_A_12 { S7_SetPoint := 'True'} : TON_TIME;
      Timer_Alarme_B_12 { S7_SetPoint := 'True'} : TON_TIME;
      Timer_Alarme_A_13 { S7_SetPoint := 'True'} : TON_TIME;
      Timer_Alarme_B_13 { S7_SetPoint := 'True'} : TON_TIME;
      Timer_Alarme_A_14 { S7_SetPoint := 'True'} : TON_TIME;
      Timer_Alarme_B_14 { S7_SetPoint := 'True'} : TON_TIME;
      Timer_Alarme_A_15 { S7_SetPoint := 'True'} : TON_TIME;
      Timer_Alarme_B_15 { S7_SetPoint := 'True'} : TON_TIME;
      Timer_Alarme_A_16 { S7_SetPoint := 'True'} : TON_TIME;
      Timer_Alarme_B_16 { S7_SetPoint := 'True'} : TON_TIME;
      Timer_Alarme_A_17 { S7_SetPoint := 'True'} : TON_TIME;
      Timer_Alarme_B_17 { S7_SetPoint := 'True'} : TON_TIME;
      Timer_Alarme_A_18 { S7_SetPoint := 'True'} : TON_TIME;
      Timer_Alarme_B_18 { S7_SetPoint := 'True'} : TON_TIME;
      Timer_Alarme_A_19 { S7_SetPoint := 'True'} : TON_TIME;
      Timer_Alarme_B_19 { S7_SetPoint := 'True'} : TON_TIME;
      Timer_Alarme_A_20 { S7_SetPoint := 'True'} : TON_TIME;
      Timer_Alarme_B_20 { S7_SetPoint := 'True'} : TON_TIME;
      Timer_Alarme_A_21 { S7_SetPoint := 'True'} : TON_TIME;
      Timer_Alarme_B_21 { S7_SetPoint := 'True'} : TON_TIME;
      Timer_Alarme_A_22 { S7_SetPoint := 'True'} : TON_TIME;
      Timer_Alarme_B_22 { S7_SetPoint := 'True'} : TON_TIME;
      Timer_Alarme_A_23 { S7_SetPoint := 'True'} : TON_TIME;
      Timer_Alarme_B_23 { S7_SetPoint := 'True'} : TON_TIME;
      Timer_Alarme_A_24 { S7_SetPoint := 'True'} : TON_TIME;
      Timer_Alarme_B_24 { S7_SetPoint := 'True'} : TON_TIME;
      Timer_Alarme_A_25 { S7_SetPoint := 'True'} : TON_TIME;
      Timer_Alarme_B_25 { S7_SetPoint := 'True'} : TON_TIME;
      Timer_Alarme_A_26 { S7_SetPoint := 'True'} : TON_TIME;
      Timer_Alarme_B_26 { S7_SetPoint := 'True'} : TON_TIME;
      Timer_Alarme_A_27 { S7_SetPoint := 'True'} : TON_TIME;
      Timer_Alarme_B_27 { S7_SetPoint := 'True'} : TON_TIME;
      Timer_Alarme_A_28 { S7_SetPoint := 'True'} : TON_TIME;
      Timer_Alarme_B_28 { S7_SetPoint := 'True'} : TON_TIME;
      Timer_Alarme_A_29 { S7_SetPoint := 'True'} : TON_TIME;
      Timer_Alarme_B_29 { S7_SetPoint := 'True'} : TON_TIME;
      Timer_Alarme_A_30 { S7_SetPoint := 'True'} : TON_TIME;
      Timer_Alarme_B_30 { S7_SetPoint := 'True'} : TON_TIME;
   END_VAR
BEGIN

REGION Network 1
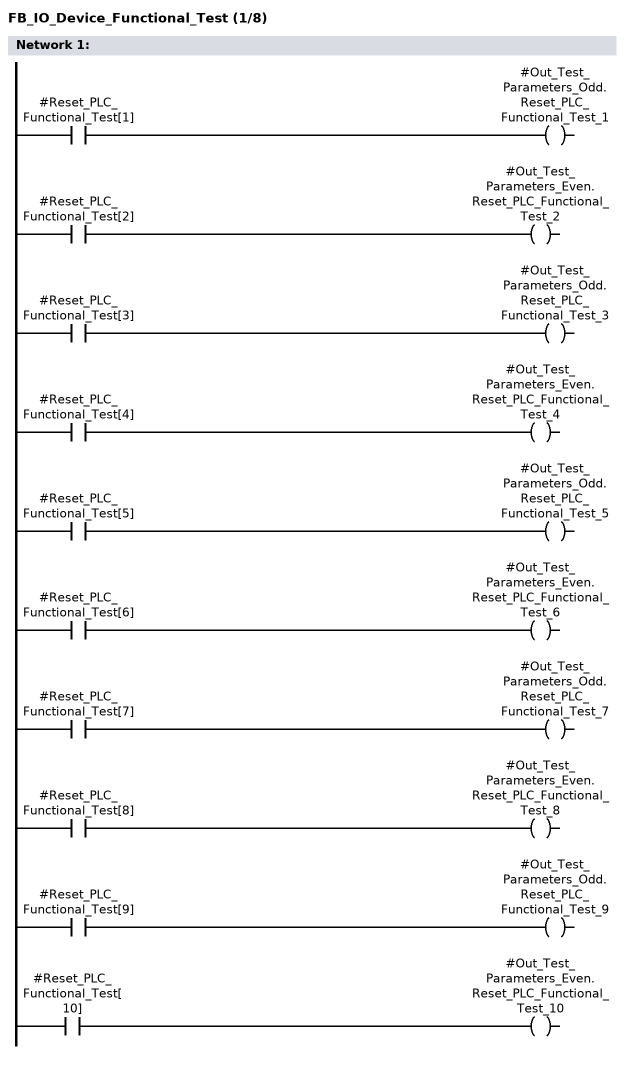
   RUNG wire#powerrail
      Contact( #Reset_PLC_Functional_Test[1] )
      Coil( #Out_Test_Parameters_Odd.Reset_PLC_Functional_Test_1 )
   END_RUNG
   RUNG wire#powerrail
      Contact( #Reset_PLC_Functional_Test[2] )
      Coil( #Out_Test_Parameters_Even.Reset_PLC_Functional_Test_2 )
   END_RUNG
   RUNG wire#powerrail
      Contact( #Reset_PLC_Functional_Test[3] )
      Coil( #Out_Test_Parameters_Odd.Reset_PLC_Functional_Test_3 )
   END_RUNG
   RUNG wire#powerrail
      Contact( #Reset_PLC_Functional_Test[4] )
      Coil( #Out_Test_Parameters_Even.Reset_PLC_Functional_Test_4 )
   END_RUNG
   RUNG wire#powerrail
      Contact( #Reset_PLC_Functional_Test[5] )
      Coil( #Out_Test_Parameters_Odd.Reset_PLC_Functional_Test_5 )
   END_RUNG
   RUNG wire#powerrail
      Contact( #Reset_PLC_Functional_Test[6] )
      Coil( #Out_Test_Parameters_Even.Reset_PLC_Functional_Test_6 )
   END_RUNG
   RUNG wire#powerrail
      Contact( #Reset_PLC_Functional_Test[7] )
      Coil( #Out_Test_Parameters_Odd.Reset_PLC_Functional_Test_7 )
   END_RUNG
   RUNG wire#powerrail
      Contact( #Reset_PLC_Functional_Test[8] )
      Coil( #Out_Test_Parameters_Even.Reset_PLC_Functional_Test_8 )
   END_RUNG
   RUNG wire#powerrail
      Contact( #Reset_PLC_Functional_Test[9] )
      Coil( #Out_Test_Parameters_Odd.Reset_PLC_Functional_Test_9 )
   END_RUNG
   RUNG wire#powerrail
      Contact( #Reset_PLC_Functional_Test[10] )
      Coil( #Out_Test_Parameters_Even.Reset_PLC_Functional_Test_10 )
   END_RUNG
   // the same network as SCL:
   #Out_Test_Parameters_Odd.Reset_PLC_Functional_Test_1 := #Reset_PLC_Functional_Test[1];
   #Out_Test_Parameters_Even.Reset_PLC_Functional_Test_2 := #Reset_PLC_Functional_Test[2];
   #Out_Test_Parameters_Odd.Reset_PLC_Functional_Test_3 := #Reset_PLC_Functional_Test[3];
   #Out_Test_Parameters_Even.Reset_PLC_Functional_Test_4 := #Reset_PLC_Functional_Test[4];
   #Out_Test_Parameters_Odd.Reset_PLC_Functional_Test_5 := #Reset_PLC_Functional_Test[5];
   #Out_Test_Parameters_Even.Reset_PLC_Functional_Test_6 := #Reset_PLC_Functional_Test[6];
   #Out_Test_Parameters_Odd.Reset_PLC_Functional_Test_7 := #Reset_PLC_Functional_Test[7];
   #Out_Test_Parameters_Even.Reset_PLC_Functional_Test_8 := #Reset_PLC_Functional_Test[8];
   #Out_Test_Parameters_Odd.Reset_PLC_Functional_Test_9 := #Reset_PLC_Functional_Test[9];
   #Out_Test_Parameters_Even.Reset_PLC_Functional_Test_10 := #Reset_PLC_Functional_Test[10];
END_REGION

REGION Network 2
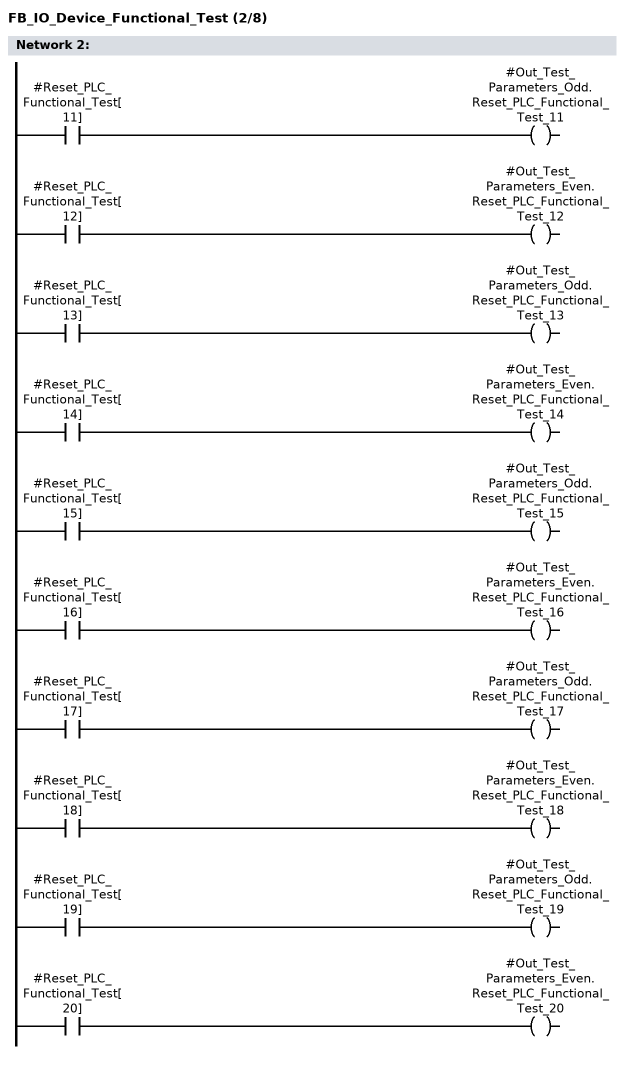
   RUNG wire#powerrail
      Contact( #Reset_PLC_Functional_Test[11] )
      Coil( #Out_Test_Parameters_Odd.Reset_PLC_Functional_Test_11 )
   END_RUNG
   RUNG wire#powerrail
      Contact( #Reset_PLC_Functional_Test[12] )
      Coil( #Out_Test_Parameters_Even.Reset_PLC_Functional_Test_12 )
   END_RUNG
   RUNG wire#powerrail
      Contact( #Reset_PLC_Functional_Test[13] )
      Coil( #Out_Test_Parameters_Odd.Reset_PLC_Functional_Test_13 )
   END_RUNG
   RUNG wire#powerrail
      Contact( #Reset_PLC_Functional_Test[14] )
      Coil( #Out_Test_Parameters_Even.Reset_PLC_Functional_Test_14 )
   END_RUNG
   RUNG wire#powerrail
      Contact( #Reset_PLC_Functional_Test[15] )
      Coil( #Out_Test_Parameters_Odd.Reset_PLC_Functional_Test_15 )
   END_RUNG
   RUNG wire#powerrail
      Contact( #Reset_PLC_Functional_Test[16] )
      Coil( #Out_Test_Parameters_Even.Reset_PLC_Functional_Test_16 )
   END_RUNG
   RUNG wire#powerrail
      Contact( #Reset_PLC_Functional_Test[17] )
      Coil( #Out_Test_Parameters_Odd.Reset_PLC_Functional_Test_17 )
   END_RUNG
   RUNG wire#powerrail
      Contact( #Reset_PLC_Functional_Test[18] )
      Coil( #Out_Test_Parameters_Even.Reset_PLC_Functional_Test_18 )
   END_RUNG
   RUNG wire#powerrail
      Contact( #Reset_PLC_Functional_Test[19] )
      Coil( #Out_Test_Parameters_Odd.Reset_PLC_Functional_Test_19 )
   END_RUNG
   RUNG wire#powerrail
      Contact( #Reset_PLC_Functional_Test[20] )
      Coil( #Out_Test_Parameters_Even.Reset_PLC_Functional_Test_20 )
   END_RUNG
   // the same network as SCL:
   #Out_Test_Parameters_Odd.Reset_PLC_Functional_Test_11 := #Reset_PLC_Functional_Test[11];
   #Out_Test_Parameters_Even.Reset_PLC_Functional_Test_12 := #Reset_PLC_Functional_Test[12];
   #Out_Test_Parameters_Odd.Reset_PLC_Functional_Test_13 := #Reset_PLC_Functional_Test[13];
   #Out_Test_Parameters_Even.Reset_PLC_Functional_Test_14 := #Reset_PLC_Functional_Test[14];
   #Out_Test_Parameters_Odd.Reset_PLC_Functional_Test_15 := #Reset_PLC_Functional_Test[15];
   #Out_Test_Parameters_Even.Reset_PLC_Functional_Test_16 := #Reset_PLC_Functional_Test[16];
   #Out_Test_Parameters_Odd.Reset_PLC_Functional_Test_17 := #Reset_PLC_Functional_Test[17];
   #Out_Test_Parameters_Even.Reset_PLC_Functional_Test_18 := #Reset_PLC_Functional_Test[18];
   #Out_Test_Parameters_Odd.Reset_PLC_Functional_Test_19 := #Reset_PLC_Functional_Test[19];
   #Out_Test_Parameters_Even.Reset_PLC_Functional_Test_20 := #Reset_PLC_Functional_Test[20];
END_REGION

REGION Network 3
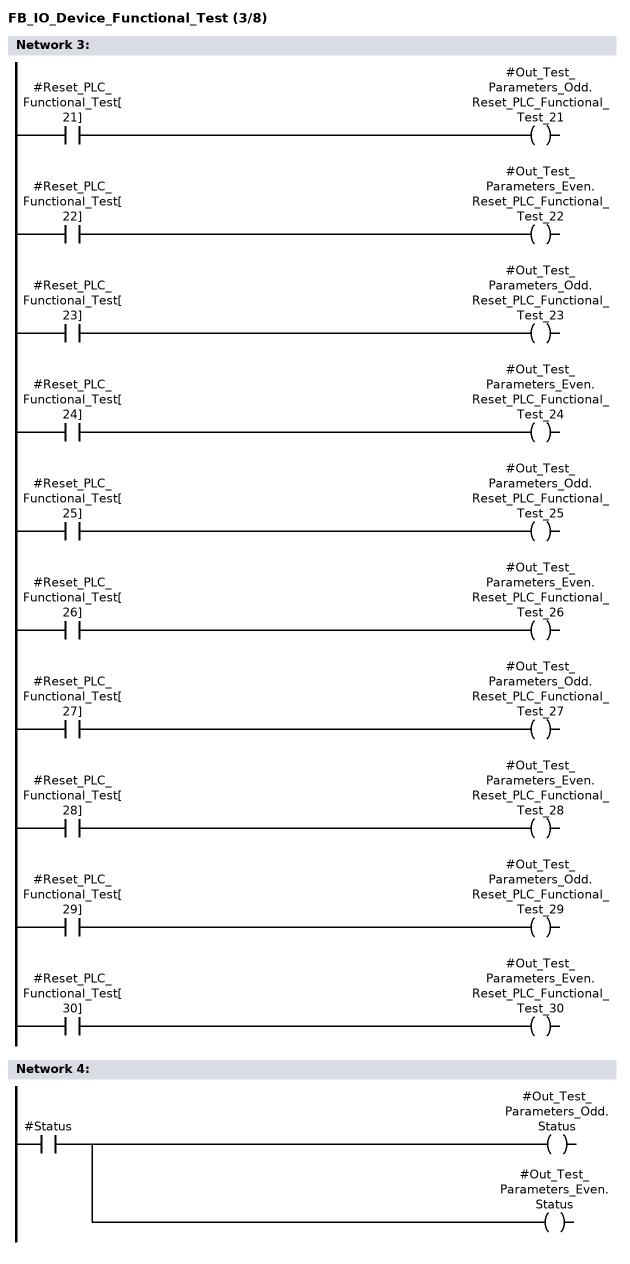
   RUNG wire#powerrail
      Contact( #Reset_PLC_Functional_Test[21] )
      Coil( #Out_Test_Parameters_Odd.Reset_PLC_Functional_Test_21 )
   END_RUNG
   RUNG wire#powerrail
      Contact( #Reset_PLC_Functional_Test[22] )
      Coil( #Out_Test_Parameters_Even.Reset_PLC_Functional_Test_22 )
   END_RUNG
   RUNG wire#powerrail
      Contact( #Reset_PLC_Functional_Test[23] )
      Coil( #Out_Test_Parameters_Odd.Reset_PLC_Functional_Test_23 )
   END_RUNG
   RUNG wire#powerrail
      Contact( #Reset_PLC_Functional_Test[24] )
      Coil( #Out_Test_Parameters_Even.Reset_PLC_Functional_Test_24 )
   END_RUNG
   RUNG wire#powerrail
      Contact( #Reset_PLC_Functional_Test[25] )
      Coil( #Out_Test_Parameters_Odd.Reset_PLC_Functional_Test_25 )
   END_RUNG
   RUNG wire#powerrail
      Contact( #Reset_PLC_Functional_Test[26] )
      Coil( #Out_Test_Parameters_Even.Reset_PLC_Functional_Test_26 )
   END_RUNG
   RUNG wire#powerrail
      Contact( #Reset_PLC_Functional_Test[27] )
      Coil( #Out_Test_Parameters_Odd.Reset_PLC_Functional_Test_27 )
   END_RUNG
   RUNG wire#powerrail
      Contact( #Reset_PLC_Functional_Test[28] )
      Coil( #Out_Test_Parameters_Even.Reset_PLC_Functional_Test_28 )
   END_RUNG
   RUNG wire#powerrail
      Contact( #Reset_PLC_Functional_Test[29] )
      Coil( #Out_Test_Parameters_Odd.Reset_PLC_Functional_Test_29 )
   END_RUNG
   RUNG wire#powerrail
      Contact( #Reset_PLC_Functional_Test[30] )
      Coil( #Out_Test_Parameters_Even.Reset_PLC_Functional_Test_30 )
   END_RUNG
   // the same network as SCL:
   #Out_Test_Parameters_Odd.Reset_PLC_Functional_Test_21 := #Reset_PLC_Functional_Test[21];
   #Out_Test_Parameters_Even.Reset_PLC_Functional_Test_22 := #Reset_PLC_Functional_Test[22];
   #Out_Test_Parameters_Odd.Reset_PLC_Functional_Test_23 := #Reset_PLC_Functional_Test[23];
   #Out_Test_Parameters_Even.Reset_PLC_Functional_Test_24 := #Reset_PLC_Functional_Test[24];
   #Out_Test_Parameters_Odd.Reset_PLC_Functional_Test_25 := #Reset_PLC_Functional_Test[25];
   #Out_Test_Parameters_Even.Reset_PLC_Functional_Test_26 := #Reset_PLC_Functional_Test[26];
   #Out_Test_Parameters_Odd.Reset_PLC_Functional_Test_27 := #Reset_PLC_Functional_Test[27];
   #Out_Test_Parameters_Even.Reset_PLC_Functional_Test_28 := #Reset_PLC_Functional_Test[28];
   #Out_Test_Parameters_Odd.Reset_PLC_Functional_Test_29 := #Reset_PLC_Functional_Test[29];
   #Out_Test_Parameters_Even.Reset_PLC_Functional_Test_30 := #Reset_PLC_Functional_Test[30];
END_REGION

REGION Network 4
   RUNG wire#powerrail
      Contact( #Status )
      wire#w1
      Coil( #Out_Test_Parameters_Odd.Status )
   END_RUNG
   RUNG wire#w1
      Coil( #Out_Test_Parameters_Even.Status )
   END_RUNG
   // the same network as SCL:
   #Out_Test_Parameters_Odd.Status := #Status;
   #Out_Test_Parameters_Even.Status := #Status;
END_REGION

REGION Network 5
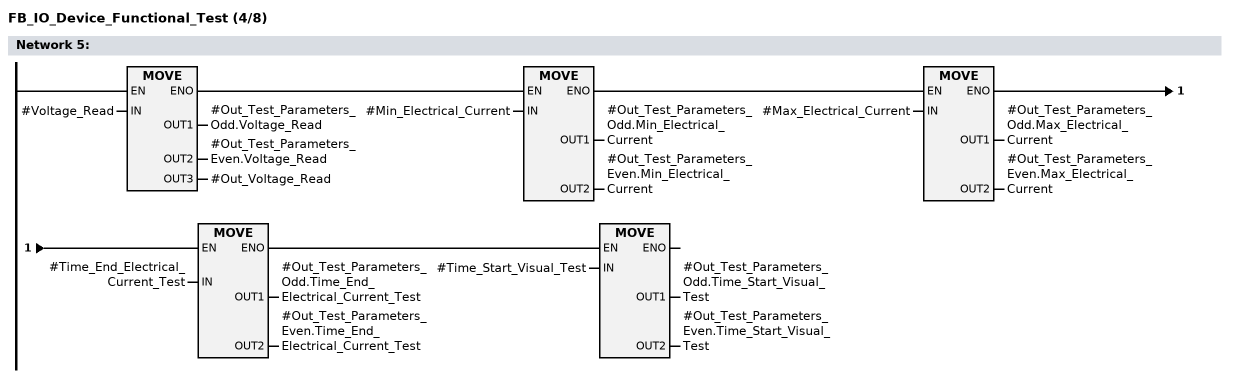
   RUNG wire#powerrail
      Move(in := #Voltage_Read, out1 => #Out_Test_Parameters_Odd.Voltage_Read, out2 => #Out_Test_Parameters_Even.Voltage_Read, out3 => #Out_Voltage_Read)
      Move(in := #Min_Electrical_Current, out1 => #Out_Test_Parameters_Odd.Min_Electrical_Current, out2 => #Out_Test_Parameters_Even.Min_Electrical_Current)
      Move(in := #Max_Electrical_Current, out1 => #Out_Test_Parameters_Odd.Max_Electrical_Current, out2 => #Out_Test_Parameters_Even.Max_Electrical_Current)
      Move(in := #Time_End_Electrical_Current_Test, out1 => #Out_Test_Parameters_Odd.Time_End_Electrical_Current_Test, out2 => #Out_Test_Parameters_Even.Time_End_Electrical_Current_Test)
      Move(in := #Time_Start_Visual_Test, out1 => #Out_Test_Parameters_Odd.Time_Start_Visual_Test, out2 => #Out_Test_Parameters_Even.Time_Start_Visual_Test)
   END_RUNG
   // the same network as SCL:
   #Out_Test_Parameters_Odd.Voltage_Read := #Voltage_Read;
   #Out_Test_Parameters_Even.Voltage_Read := #Voltage_Read;
   #Out_Voltage_Read := #Voltage_Read;
   #Out_Test_Parameters_Odd.Min_Electrical_Current := #Min_Electrical_Current;
   #Out_Test_Parameters_Even.Min_Electrical_Current := #Min_Electrical_Current;
   #Out_Test_Parameters_Odd.Max_Electrical_Current := #Max_Electrical_Current;
   #Out_Test_Parameters_Even.Max_Electrical_Current := #Max_Electrical_Current;
   #Out_Test_Parameters_Odd.Time_End_Electrical_Current_Test := #Time_End_Electrical_Current_Test;
   #Out_Test_Parameters_Even.Time_End_Electrical_Current_Test := #Time_End_Electrical_Current_Test;
   #Out_Test_Parameters_Odd.Time_Start_Visual_Test := #Time_Start_Visual_Test;
   #Out_Test_Parameters_Even.Time_Start_Visual_Test := #Time_Start_Visual_Test;
END_REGION

